   t1[22376] := -0.0600096;
   t1[22377] := -0.0732072;
   t1[22378] := -0.0857643;
   t1[22379] := -0.097705;
   t1[22380] := -0.1090593;
   t1[22381] := -0.1198572;
   t1[22382] := -0.130129;
   t1[22383] := -0.1399046;
   t1[22384] := -0.1492141;
   t1[22385] := -0.1580877;
   t1[22386] := -0.1665554;
   t1[22387] := -0.1746473;
   t1[22388] := -0.1823935;
   t1[22389] := -0.189824;
   t1[22390] := -0.196969;
   t1[22391] := -0.2038585;
   t1[22392] := -0.2105227;
   t1[22393] := -0.2169916;
   t1[22394] := -0.2232952;
   t1[22395] := -0.2294637;
   t1[22396] := -0.2355272;
   t1[22397] := -0.2415041;
   t1[22398] := -0.2473547;
   t1[22399] := -0.2530213;
   w2[0] := 0.3822261;
   w2[1] := 0.6735258;
   w2[2] := 0.4999258;
   w2[3] := 0.0709843;
   w2[4] := 0.4040336;
   w2[5] := -0.3168498;
   w2[6] := -0.5318553;
   w2[7] := -0.3348889;
   w2[8] := 0.5234552;
   w2[9] := 0.3241403;
   w2[10] := -0.6014917;
   w2[11] := -0.2869324;
   w2[12] := -0.0813316;
   w2[13] := 0.2735443;
   w2[14] := -0.5975453;
   w2[15] := -0.3671676;
   w2[16] := 0.1604395;
   w2[17] := 0.6218057;
   w2[18] := -0.535407;
   w2[19] := -0.428839;
   w2[20] := 0.4432988;
   w2[21] := -0.1195226;
   w2[22] := -0.1593684;
   w2[23] := -0.4208567;
   w2[24] := -0.0164311;
   w2[25] := 0.1177106;
   w2[26] := -0.1915699;
   w2[27] := -0.2585908;
   w2[28] := 0.7388805;
   w2[29] := 0.7177937;
   w2[30] := 0.9066412;
   w2[31] := -0.3313666;
   w2[32] := -0.5566195;
   w2[33] := 0.1009696;
   w2[34] := 0.7024983;
   w2[35] := -0.0061407;
   w2[36] := 0.9221094;
   w2[37] := 0.9728315;
   w2[38] := 0.7287791;
   w2[39] := 0.1011917;
   w2[40] := 0.1708561;
   w2[41] := 0.0181266;
   w2[42] := -0.3799455;
   w2[43] := -0.2221509;
   w2[44] := -0.2996568;
   w2[45] := 0.1856399;
   w2[46] := -0.2363337;
   w2[47] := 0.3469633;
   w2[48] := -0.3170906;
   w2[49] := -0.3010724;
   w2[50] := -0.4463713;
   w2[51] := 0.4818622;
   w2[52] := -0.2695292;
   w2[53] := -0.4620254;
   w2[54] := 0.0533027;
   w2[55] := -0.395156;
   w2[56] := 0.0408355;
   w2[57] := -0.2507218;
   w2[58] := 0.0280879;
   w2[59] := 0.0458854;
   w2[60] := -0.0139494;
   w2[61] := 0.0098419;
   w2[62] := -0.4868755;
   w2[63] := 0.1032088;
   w2[64] := 0.1231787;
   w2[65] := 0.5223995;
   w2[66] := 0.4042619;
   w2[67] := 0.2341684;
   w2[68] := -0.2304757;
   w2[69] := 0.0635033;
   w2[70] := -0.3774453;
   w2[71] := -0.4428134;
   w2[72] := -0.0484126;
   w2[73] := 0.2895669;
   w2[74] := -0.6764416;
   w2[75] := -0.3088431;
   w2[76] := 0.4827037;
   w2[77] := 0.0691548;
   w2[78] := 0.4661854;
   w2[79] := 0.1204736;
   w2[80] := -0.4872637;
   w2[81] := -0.0951735;
   w2[82] := -0.0189593;
   w2[83] := -0.1372051;
   w2[84] := -0.9140335;
   w2[85] := -0.8600995;
   w2[86] := -1.056187;
   w2[87] := -0.5128109;
   w2[88] := -0.7898985;
   w2[89] := -0.5083115;
   w2[90] := -0.5282256;
   w2[91] := -0.4263123;
   w2[92] := -1.016044;
   w2[93] := -0.0212463;
   w2[94] := 0.6550046;
   w2[95] := 0.4706961;
   w2[96] := -0.1141442;
   w2[97] := -0.2175039;
   w2[98] := -0.2840221;
   w2[99] := -0.3306261;
   w2[100] := -0.2441688;
   w2[101] := 0.3605514;
   w2[102] := -0.3955784;
   w2[103] := 0.0529358;
   w2[104] := 0.3398173;
   w2[105] := 0.3715278;
   w2[106] := 0.429172;
   w2[107] := 0.4002611;
   w2[108] := -0.2264336;
   w2[109] := 0.312763;
   w2[110] := 0.5647593;
   w2[111] := 0.0224205;
   w2[112] := -0.5216327;
   w2[113] := -0.2093005;
   w2[114] := -0.3824884;
   w2[115] := -0.0496232;
   w2[116] := -0.0204715;
   w2[117] := 0.3446302;
   w2[118] := -0.1566623;
   w2[119] := -0.1314349;
   w2[120] := -0.3364701;
   w2[121] := -0.5365704;
   w2[122] := -0.3706124;
   w2[123] := -0.2384351;
   w2[124] := 0.2599077;
   w2[125] := 0.0878742;
   w2[126] := -0.1167608;
   w2[127] := 0.4445257;
   w2[128] := 0.0472859;
   w2[129] := -0.2039315;
   w2[130] := -0.0123044;
   w2[131] := 0.5347427;
   w2[132] := -0.4565654;
   w2[133] := -0.1309683;
   w2[134] := -0.1916631;
   w2[135] := -0.0229556;
   w2[136] := -0.1463313;
   w2[137] := 0.0884493;
   w2[138] := -0.1268248;
   w2[139] := 0.1727386;
   w2[140] := 0.1864566;
   w2[141] := 0.0450289;
   w2[142] := 0.2544484;
   w2[143] := -0.1416016;
   w2[144] := -0.1781151;
   w2[145] := -0.1914191;
   w2[146] := 0.3022377;
   w2[147] := 0.2656204;
   w2[148] := 0.135544;
   w2[149] := 0.5225624;
   w2[150] := 0.8165789;
   w2[151] := 0.3793563;
   w2[152] := -0.1251971;
   w2[153] := -0.032513;
   w2[154] := -0.1753309;
   w2[155] := -0.429324;
   w2[156] := -0.4619711;
   w2[157] := 0.3961401;
   w2[158] := -0.6358346;
   w2[159] := 0.531637;
   w2[160] := 0.2908633;
   w2[161] := 0.2183272;
   w2[162] := 0.3942987;
   w2[163] := 0.3020125;
   w2[164] := -0.4793546;
   w2[165] := 0.0537859;
   w2[166] := 0.2855184;
   w2[167] := -0.2678719;
   w2[168] := 0.3169011;
   w2[169] := 0.0269058;
   w2[170] := 0.139307;
   w2[171] := 0.2074015;
   w2[172] := 0.044378;
   w2[173] := 0.3336064;
   w2[174] := -0.1919886;
   w2[175] := 0.0043234;
   w2[176] := 0.5604227;
   w2[177] := -0.1127777;
   w2[178] := -0.3165137;
   w2[179] := 0.2200206;
   w2[180] := -0.2163805;
   w2[181] := -0.239696;
   w2[182] := 0.1728129;
   w2[183] := -0.1887252;
   w2[184] := 0.2727011;
   w2[185] := 0.1560453;
   w2[186] := 0.457509;
   w2[187] := -0.2272316;
   w2[188] := 0.3077642;
   w2[189] := 0.06774;
   w2[190] := -0.050842;
   w2[191] := 0.0844207;
   w2[192] := 0.2612096;
   w2[193] := -0.0461612;
   w2[194] := 0.196588;
   w2[195] := 0.1832603;
   w2[196] := -0.1259902;
   w2[197] := 0.4958175;
   w2[198] := 0.3578667;
   w2[199] := -0.2289235;
   w2[200] := 0.0412198;
   w2[201] := -0.1472023;
   w2[202] := 0.5003238;
   w2[203] := 0.2104491;
   w2[204] := -0.3506398;
   w2[205] := -0.7278167;
   w2[206] := -0.1053378;
   w2[207] := -0.6664331;
   w2[208] := 0.3304765;
   w2[209] := 0.1904697;
   w2[210] := -0.5255481;
   w2[211] := 0.3779066;
   w2[212] := 0.575013;
   w2[213] := -0.4405918;
   w2[214] := 0.0437819;
   w2[215] := 0.0799071;
   w2[216] := -0.3873571;
   w2[217] := -0.1107465;
   w2[218] := -0.2144487;
   w2[219] := -0.452094;
   w2[220] := -0.0942226;
   w2[221] := -0.1042965;
   w2[222] := -0.0900685;
   w2[223] := -0.0358909;
   w2[224] := 0.5961101;
   w2[225] := -0.0502036;
   w2[226] := -0.205787;
   w2[227] := 0.1793782;
   w2[228] := 0.0139435;
   w2[229] := 0.140426;
   w2[230] := -0.1710399;
   w2[231] := -0.1097762;
   w2[232] := 0.6955358;
   w2[233] := -0.0941478;
   w2[234] := -0.6882815;
   w2[235] := -0.2339452;
   w2[236] := -0.5887371;
   w2[237] := 0.0302498;
   w2[238] := 0.2707806;
   w2[239] := -0.6653628;
   w2[240] := 0.3887634;
   w2[241] := 0.1627363;
   w2[242] := 0.0122889;
   w2[243] := -0.4034282;
   w2[244] := 0.3380547;
   w2[245] := -0.0177897;
   w2[246] := -0.1635698;
   w2[247] := -0.1298062;
   w2[248] := 0.2896215;
   w2[249] := 0.1131524;
   w2[250] := -0.2054364;
   w2[251] := 0.0131579;
   w2[252] := -0.890228;
   w2[253] := -0.6914336;
   w2[254] := -0.8277874;
   w2[255] := 0.254033;
   w2[256] := 0.179194;
   w2[257] := 0.0266804;
   w2[258] := -0.1867425;
   w2[259] := 0.1680747;
   w2[260] := -1.05107;
   w2[261] := -0.5665534;
   w2[262] := -0.1247267;
   w2[263] := -0.053494;
   w2[264] := 0.23726;
   w2[265] := -0.584154;
   w2[266] := -0.2938985;
   w2[267] := 0.1965791;
   w2[268] := 0.5103638;
   w2[269] := -0.0550255;
   w2[270] := -1.126066;
   w2[271] := 0.0735265;
   w2[272] := -0.2777269;
   w2[273] := 0.3135782;
   w2[274] := 0.1041824;
   w2[275] := -0.1324059;
   w2[276] := -0.3669493;
   w2[277] := -0.2885313;
   w2[278] := -0.367729;
   w2[279] := 0.1541151;
   w2[280] := 0.1346243;
   w2[281] := 0.6931639;
   w2[282] := 0.3574378;
   w2[283] := -0.1421183;
   w2[284] := 0.2825844;
   w2[285] := 0.0992049;
   w2[286] := 0.3324718;
   w2[287] := 0.168798;
   w2[288] := 0.1662632;
   w2[289] := -0.5125447;
   w2[290] := 0.1457812;
   w2[291] := -0.2258452;
   w2[292] := -0.2428768;
   w2[293] := 0.2717957;
   w2[294] := 0.0867224;
   w2[295] := -0.2496022;
   w2[296] := 0.1867056;
   w2[297] := -0.4031086;
   w2[298] := 0.4832774;
   w2[299] := 0.2478154;
   w2[300] := 0.0475016;
   w2[301] := -0.1532699;
   w2[302] := -0.6021184;
   w2[303] := -0.4835578;
   w2[304] := 0.348039;
   w2[305] := -0.0061014;
   w2[306] := 0.2888969;
   w2[307] := 0.0215752;
   w2[308] := 0.0208341;
   w2[309] := 0.5199659;
   w2[310] := 0.3490263;
   w2[311] := -0.0288161;
   w2[312] := -0.068543;
   w2[313] := -0.1182679;
   w2[314] := 0.3420109;
   w2[315] := -0.0353185;
   w2[316] := -0.1071727;
   w2[317] := -0.7671919;
   w2[318] := -0.3097001;
   w2[319] := 0.0119445;
   w2[320] := 0.1677119;
   w2[321] := -0.0187103;
   w2[322] := -0.0632623;
   w2[323] := 0.3558021;
   w2[324] := 0.4361037;
   w2[325] := -0.5477799;
   w2[326] := 0.1640894;
   w2[327] := 0.3476633;
   w2[328] := -0.2296589;
   w2[329] := -0.0005878;
   w2[330] := -0.1486427;
   w2[331] := -0.1145124;
   w2[332] := 0.1935411;
   w2[333] := -0.0498571;
   w2[334] := 0.007102;
   w2[335] := 0.1442345;
   w2[336] := -0.7647343;
   w2[337] := -0.7446802;
   w2[338] := -0.8727151;
   w2[339] := 0.3649753;
   w2[340] := 0.182284;
   w2[341] := 0.2168968;
   w2[342] := -0.3110866;
   w2[343] := 0.2285281;
   w2[344] := -0.8572159;
   w2[345] := -0.253249;
   w2[346] := -0.1099993;
   w2[347] := -0.1176312;
   w2[348] := 0.3110442;
   w2[349] := -0.0493409;
   w2[350] := 0.0371198;
   w2[351] := 0.2336326;
   w2[352] := 0.2238284;
   w2[353] := -0.0283122;
   w2[354] := -0.1704783;
   w2[355] := 0.0574998;
   w2[356] := -0.2733924;
   w2[357] := 0.0665076;
   w2[358] := 0.0320759;
   w2[359] := -0.1596949;
   w2[360] := -0.2385386;
   w2[361] := -0.2472534;
   w2[362] := -0.1323308;
   w2[363] := 0.1628101;
   w2[364] := 0.4503315;
   w2[365] := 0.1501646;
   w2[366] := 0.1143262;
   w2[367] := 0.023902;
   w2[368] := 0.0073025;
   w2[369] := 0.1456288;
   w2[370] := -0.3334046;
   w2[371] := 0.0482971;
   w2[372] := 0.4867398;
   w2[373] := -0.4917139;
   w2[374] := -0.6253324;
   w2[375] := -0.1267435;
   w2[376] := -0.2428251;
   w2[377] := -0.2196695;
   w2[378] := 0.1073758;
   w2[379] := 0.0506342;
   w2[380] := 0.4630886;
   w2[381] := -0.1982542;
   w2[382] := 0.3006389;
   w2[383] := -0.1852189;
   w2[384] := 0.1438557;
   w2[385] := 0.2112408;
   w2[386] := -0.1989525;
   w2[387] := -0.5165743;
   w2[388] := 0.2818699;
   w2[389] := 0.1988503;
   w2[390] := 0.0899179;
   w2[391] := 0.0992274;
   w2[392] := 0.3425773;
   w2[393] := -0.0475926;
   w2[394] := 0.0767343;
   w2[395] := 0.0394692;
   w2[396] := 0.1684201;
   w2[397] := -0.1340467;
   w2[398] := -0.3633062;
   w2[399] := -0.3210598;
   w2[400] := 0.5503753;
   w2[401] := 0.2680424;
   w2[402] := -0.2979992;
   w2[403] := -0.3373846;
   w2[404] := -0.2860682;
   w2[405] := 0.0260232;
   w2[406] := -0.1706583;
   w2[407] := -0.4802254;
   w2[408] := 0.1432097;
   w2[409] := 0.2762946;
   w2[410] := -0.3853753;
   w2[411] := -0.4026088;
   w2[412] := 0.3293981;
   w2[413] := 0.031134;
   w2[414] := 0.1150283;
   w2[415] := 0.032845;
   w2[416] := 0.1377832;
   w2[417] := 0.2112923;
   w2[418] := 0.0084318;
   w2[419] := 0.0693316;
   w2[420] := 0.0293756;
   w2[421] := 0.1045898;
   w2[422] := 0.2854653;
   w2[423] := 0.0997073;
   w2[424] := 0.1003512;
   w2[425] := -0.0351206;
   w2[426] := 0.4399726;
   w2[427] := 0.2780291;
   w2[428] := -0.0804132;
   w2[429] := 0.7397832;
   w2[430] := 0.7269561;
   w2[431] := 0.2094024;
   w2[432] := -0.2141474;
   w2[433] := 0.2012126;
   w2[434] := -0.2318728;
   w2[435] := -0.1762547;
   w2[436] := -0.0704646;
   w2[437] := 0.2301458;
   w2[438] := -0.0323121;
   w2[439] := 0.1872706;
   w2[440] := 0.4350786;
   w2[441] := 0.266441;
   w2[442] := 0.2541361;
   w2[443] := 0.1549129;
   w2[444] := -0.1279981;
   w2[445] := -0.1567508;
   w2[446] := 0.1148285;
   w2[447] := -0.2802774;
   g4[0] := -3.0;
   g4[1] := -2.877551;
   g4[2] := -2.755102;
   g4[3] := -2.632653;
   g4[4] := -2.510204;
   g4[5] := -2.387755;
   g4[6] := -2.265306;
   g4[7] := -2.142857;
   g4[8] := -2.020408;
   g4[9] := -1.897959;
   g4[10] := -1.77551;
   g4[11] := -1.653061;
   g4[12] := -1.530612;
   g4[13] := -1.408163;
   g4[14] := -1.285714;
   g4[15] := -1.163265;
   g4[16] := -1.040816;
   g4[17] := -0.9183673;
   g4[18] := -0.7959184;
   g4[19] := -0.6734694;
   g4[20] := -0.5510204;
   g4[21] := -0.4285714;
   g4[22] := -0.3061224;
   g4[23] := -0.1836735;
   g4[24] := -0.0612245;
   g4[25] := 0.0612245;
   g4[26] := 0.1836735;
   g4[27] := 0.3061224;
   g4[28] := 0.4285714;
   g4[29] := 0.5510204;
   g4[30] := 0.6734694;
   g4[31] := 0.7959184;
   g4[32] := 0.9183673;
   g4[33] := 1.040816;
   g4[34] := 1.163265;
   g4[35] := 1.285714;
   g4[36] := 1.408163;
   g4[37] := 1.530612;
   g4[38] := 1.653061;
   g4[39] := 1.77551;
   g4[40] := 1.897959;
   g4[41] := 2.020408;
   g4[42] := 2.142857;
   g4[43] := 2.265306;
   g4[44] := 2.387755;
   g4[45] := 2.510204;
   g4[46] := 2.632653;
   g4[47] := 2.755102;
   g4[48] := 2.877551;
   g4[49] := 3.0;
   t5[0] := 0.0969458;
   t5[1] := 0.0975005;
   t5[2] := 0.0980442;
   t5[3] := 0.0985769;
   t5[4] := 0.0990984;
   t5[5] := 0.0996084;
   t5[6] := 0.1001068;
   t5[7] := 0.1005933;
   t5[8] := 0.1010678;
   t5[9] := 0.1015302;
   t5[10] := 0.1019801;
   t5[11] := 0.1024174;
   t5[12] := 0.102842;
   t5[13] := 0.1032536;
   t5[14] := 0.1036521;
   t5[15] := 0.1040372;
   t5[16] := 0.1044088;
   t5[17] := 0.1047666;
   t5[18] := 0.1051106;
   t5[19] := 0.1054404;
   t5[20] := 0.105756;
   t5[21] := 0.1060571;
   t5[22] := 0.1063435;
   t5[23] := 0.1066151;
   t5[24] := 0.1068716;
   t5[25] := 0.1071129;
   t5[26] := 0.1073388;
   t5[27] := 0.107549;
   t5[28] := 0.1077435;
   t5[29] := 0.1079219;
   t5[30] := 0.1080842;
   t5[31] := 0.1082301;
   t5[32] := 0.1083595;
   t5[33] := 0.1084721;
   t5[34] := 0.1085678;
   t5[35] := 0.1086466;
   t5[36] := 0.1087088;
   t5[37] := 0.1087546;
   t5[38] := 0.1087841;
   t5[39] := 0.1087976;
   t5[40] := 0.1087953;
   t5[41] := 0.1087774;
   t5[42] := 0.1087441;
   t5[43] := 0.1086956;
   t5[44] := 0.1086322;
   t5[45] := 0.1085539;
   t5[46] := 0.1084611;
   t5[47] := 0.1083539;
   t5[48] := 0.1082325;
   t5[49] := 0.1080972;
   t5[50] := 0.0692292;
   t5[51] := 0.0688175;
   t5[52] := 0.0684027;
   t5[53] := 0.0679847;
   t5[54] := 0.0675634;
   t5[55] := 0.0671384;
   t5[56] := 0.0667096;
   t5[57] := 0.0662769;
   t5[58] := 0.0658399;
   t5[59] := 0.0653986;
   t5[60] := 0.0649527;
   t5[61] := 0.0645021;
   t5[62] := 0.0640465;
   t5[63] := 0.0635857;
   t5[64] := 0.0631196;
   t5[65] := 0.062648;
   t5[66] := 0.0621706;
   t5[67] := 0.0616873;
   t5[68] := 0.0611979;
   t5[69] := 0.0607022;
   t5[70] := 0.0601999;
   t5[71] := 0.059691;
   t5[72] := 0.0591752;
   t5[73] := 0.0586522;
   t5[74] := 0.058122;
   t5[75] := 0.0575843;
   t5[76] := 0.057039;
   t5[77] := 0.0564858;
   t5[78] := 0.0559245;
   t5[79] := 0.055355;
   t5[80] := 0.054777;
   t5[81] := 0.0541904;
   t5[82] := 0.0535949;
   t5[83] := 0.0529904;
   t5[84] := 0.0523768;
   t5[85] := 0.051754;
   t5[86] := 0.0511223;
   t5[87] := 0.050482;
   t5[88] := 0.0498332;
   t5[89] := 0.0491762;
   t5[90] := 0.0485112;
   t5[91] := 0.0478384;
   t5[92] := 0.0471581;
   t5[93] := 0.0464705;
   t5[94] := 0.0457757;
   t5[95] := 0.0450742;
   t5[96] := 0.0443659;
   t5[97] := 0.0436513;
   t5[98] := 0.0429304;
   t5[99] := 0.0422036;
   t5[100] := 0.0769506;
   t5[101] := 0.0760873;
   t5[102] := 0.0752231;
   t5[103] := 0.074358;
   t5[104] := 0.0734922;
   t5[105] := 0.0726259;
   t5[106] := 0.0717593;
   t5[107] := 0.0708925;
   t5[108] := 0.0700258;
   t5[109] := 0.0691593;
   t5[110] := 0.0682932;
   t5[111] := 0.0674276;
   t5[112] := 0.0665628;
   t5[113] := 0.0656989;
   t5[114] := 0.0648361;
   t5[115] := 0.0639746;
   t5[116] := 0.0631145;
   t5[117] := 0.0622561;
   t5[118] := 0.0613995;
   t5[119] := 0.0605449;
   t5[120] := 0.0596924;
   t5[121] := 0.0588422;
   t5[122] := 0.0579946;
   t5[123] := 0.0571497;
   t5[124] := 0.0563077;
   t5[125] := 0.0554687;
   t5[126] := 0.0546329;
   t5[127] := 0.0538006;
   t5[128] := 0.0529718;
   t5[129] := 0.0521468;
   t5[130] := 0.0513257;
   t5[131] := 0.0505087;
   t5[132] := 0.049696;
   t5[133] := 0.0488878;
   t5[134] := 0.0480843;
   t5[135] := 0.0472854;
   t5[136] := 0.0464911;
   t5[137] := 0.0457015;
   t5[138] := 0.0449164;
   t5[139] := 0.0441359;
   t5[140] := 0.0433598;
   t5[141] := 0.0425883;
   t5[142] := 0.0418212;
   t5[143] := 0.0410585;
   t5[144] := 0.0403002;
   t5[145] := 0.0395462;
   t5[146] := 0.0387965;
   t5[147] := 0.0380511;
   t5[148] := 0.03731;
   t5[149] := 0.036573;
   t5[150] := 0.0185666;
   t5[151] := 0.018039;
   t5[152] := 0.0175079;
   t5[153] := 0.0169733;
   t5[154] := 0.0164355;
   t5[155] := 0.0158946;
   t5[156] := 0.0153508;
   t5[157] := 0.0148043;
   t5[158] := 0.0142552;
   t5[159] := 0.0137036;
   t5[160] := 0.0131499;
   t5[161] := 0.012594;
   t5[162] := 0.0120363;
   t5[163] := 0.0114768;
   t5[164] := 0.0109158;
   t5[165] := 0.0103533;
   t5[166] := 0.0097896;
   t5[167] := 0.0092249;
   t5[168] := 0.0086592;
   t5[169] := 0.0080928;
   t5[170] := 0.0075258;
   t5[171] := 0.0069585;
   t5[172] := 0.0063908;
   t5[173] := 0.0058232;
   t5[174] := 0.0052556;
   t5[175] := 0.0046883;
   t5[176] := 0.0041214;
   t5[177] := 0.0035551;
   t5[178] := 0.0029896;
   t5[179] := 0.002425;
   t5[180] := 0.0018615;
   t5[181] := 0.0012993;
   t5[182] := 0.0007385;
   t5[183] := 0.0001793;
   t5[184] := -0.0003781;
   t5[185] := -0.0009336;
   t5[186] := -0.0014869;
   t5[187] := -0.002038;
   t5[188] := -0.0025867;
   t5[189] := -0.0031328;
   t5[190] := -0.0036761;
   t5[191] := -0.0042165;
   t5[192] := -0.0047537;
   t5[193] := -0.0052877;
   t5[194] := -0.0058183;
   t5[195] := -0.0063453;
   t5[196] := -0.0068684;
   t5[197] := -0.0073877;
   t5[198] := -0.0079029;
   t5[199] := -0.0084138;
   t5[200] := -0.0480992;
   t5[201] := -0.0461759;
   t5[202] := -0.0442379;
   t5[203] := -0.0422851;
   t5[204] := -0.0403176;
   t5[205] := -0.0383352;
   t5[206] := -0.0363378;
   t5[207] := -0.0343254;
   t5[208] := -0.0322979;
   t5[209] := -0.0302553;
   t5[210] := -0.0281974;
   t5[211] := -0.0261242;
   t5[212] := -0.0240356;
   t5[213] := -0.0219317;
   t5[214] := -0.0198121;
   t5[215] := -0.017677;
   t5[216] := -0.0155263;
   t5[217] := -0.0133598;
   t5[218] := -0.0111775;
   t5[219] := -0.0089794;
   t5[220] := -0.0067653;
   t5[221] := -0.0045353;
   t5[222] := -0.0022891;
   t5[223] := -2.68E-05;
   t5[224] := 0.0022517;
   t5[225] := 0.0045464;
   t5[226] := 0.0068576;
   t5[227] := 0.0091852;
   t5[228] := 0.0115292;
   t5[229] := 0.0138899;
   t5[230] := 0.0162671;
   t5[231] := 0.0186611;
   t5[232] := 0.0210719;
   t5[233] := 0.0234995;
   t5[234] := 0.025944;
   t5[235] := 0.028405;
   t5[236] := 0.0308823;
   t5[237] := 0.0333751;
   t5[238] := 0.035883;
   t5[239] := 0.0384056;
   t5[240] := 0.0409424;
   t5[241] := 0.0434929;
   t5[242] := 0.0460565;
   t5[243] := 0.0486329;
   t5[244] := 0.0512215;
   t5[245] := 0.0538219;
   t5[246] := 0.0564335;
   t5[247] := 0.059056;
   t5[248] := 0.0616887;
   t5[249] := 0.0643312;
   t5[250] := 0.0416106;
   t5[251] := 0.0407638;
   t5[252] := 0.039913;
   t5[253] := 0.0390582;
   t5[254] := 0.0381993;
   t5[255] := 0.0373361;
   t5[256] := 0.0364686;
   t5[257] := 0.0355967;
   t5[258] := 0.0347203;
   t5[259] := 0.0338393;
   t5[260] := 0.0329536;
   t5[261] := 0.0320632;
   t5[262] := 0.031168;
   t5[263] := 0.0302678;
   t5[264] := 0.0293625;
   t5[265] := 0.0284521;
   t5[266] := 0.0275366;
   t5[267] := 0.0266157;
   t5[268] := 0.0256895;
   t5[269] := 0.0247577;
   t5[270] := 0.0238204;
   t5[271] := 0.0228775;
   t5[272] := 0.0219288;
   t5[273] := 0.0209743;
   t5[274] := 0.0200138;
   t5[275] := 0.0190474;
   t5[276] := 0.0180748;
   t5[277] := 0.0170961;
   t5[278] := 0.0161111;
   t5[279] := 0.0151197;
   t5[280] := 0.0141218;
   t5[281] := 0.0131174;
   t5[282] := 0.0121064;
   t5[283] := 0.0110886;
   t5[284] := 0.0100641;
   t5[285] := 0.0090329;
   t5[286] := 0.0079953;
   t5[287] := 0.0069515;
   t5[288] := 0.005902;
   t5[289] := 0.0048468;
   t5[290] := 0.0037862;
   t5[291] := 0.0027206;
   t5[292] := 0.0016502;
   t5[293] := 0.0005753;
   t5[294] := -0.000504;
   t5[295] := -0.0015873;
   t5[296] := -0.0026743;
   t5[297] := -0.0037649;
   t5[298] := -0.0048587;
   t5[299] := -0.0059555;
   t5[300] := 0.040686;
   t5[301] := 0.0380326;
   t5[302] := 0.0353805;
   t5[303] := 0.0327302;
   t5[304] := 0.0300825;
   t5[305] := 0.0274376;
   t5[306] := 0.0247961;
   t5[307] := 0.0221584;
   t5[308] := 0.0195253;
   t5[309] := 0.016897;
   t5[310] := 0.0142741;
   t5[311] := 0.0116571;
   t5[312] := 0.0090466;
   t5[313] := 0.006443;
   t5[314] := 0.0038467;
   t5[315] := 0.0012584;
   t5[316] := -0.0013215;
   t5[317] := -0.0038925;
   t5[318] := -0.0064541;
   t5[319] := -0.0090057;
   t5[320] := -0.0115469;
   t5[321] := -0.0140773;
   t5[322] := -0.0165961;
   t5[323] := -0.0191031;
   t5[324] := -0.0215977;
   t5[325] := -0.0240793;
   t5[326] := -0.0265474;
   t5[327] := -0.0290017;
   t5[328] := -0.0314415;
   t5[329] := -0.0338664;
   t5[330] := -0.0362759;
   t5[331] := -0.0386694;
   t5[332] := -0.0410465;
   t5[333] := -0.0434067;
   t5[334] := -0.0457494;
   t5[335] := -0.0480745;
   t5[336] := -0.050382;
   t5[337] := -0.0526716;
   t5[338] := -0.0549433;
   t5[339] := -0.0571972;
   t5[340] := -0.059433;
   t5[341] := -0.0616507;
   t5[342] := -0.0638503;
   t5[343] := -0.0660316;
   t5[344] := -0.0681946;
   t5[345] := -0.0703393;
   t5[346] := -0.0724654;
   t5[347] := -0.074573;
   t5[348] := -0.076662;
   t5[349] := -0.0787324;
   t5[350] := 0.0090538;
   t5[351] := 0.00985;
   t5[352] := 0.0106394;
   t5[353] := 0.0114219;
   t5[354] := 0.0121974;
   t5[355] := 0.0129658;
   t5[356] := 0.0137272;
   t5[357] := 0.0144813;
   t5[358] := 0.0152283;
   t5[359] := 0.015968;
   t5[360] := 0.0167005;
   t5[361] := 0.0174255;
   t5[362] := 0.0181432;
   t5[363] := 0.0188533;
   t5[364] := 0.019556;
   t5[365] := 0.020251;
   t5[366] := 0.0209385;
   t5[367] := 0.0216182;
   t5[368] := 0.0222903;
   t5[369] := 0.0229545;
   t5[370] := 0.0236109;
   t5[371] := 0.0242594;
   t5[372] := 0.0248999;
   t5[373] := 0.0255325;
   t5[374] := 0.026157;
   t5[375] := 0.0267733;
   t5[376] := 0.0273816;
   t5[377] := 0.0279816;
   t5[378] := 0.0285733;
   t5[379] := 0.0291567;
   t5[380] := 0.0297317;
   t5[381] := 0.0302983;
   t5[382] := 0.0308565;
   t5[383] := 0.0314061;
   t5[384] := 0.0319471;
   t5[385] := 0.0324795;
   t5[386] := 0.0330033;
   t5[387] := 0.0335185;
   t5[388] := 0.0340251;
   t5[389] := 0.0345232;
   t5[390] := 0.0350126;
   t5[391] := 0.0354935;
   t5[392] := 0.0359658;
   t5[393] := 0.0364295;
   t5[394] := 0.0368846;
   t5[395] := 0.0373312;
   t5[396] := 0.0377692;
   t5[397] := 0.0381986;
   t5[398] := 0.0386195;
   t5[399] := 0.0390318;
   t5[400] := 0.0821998;
   t5[401] := 0.0816142;
   t5[402] := 0.0810245;
   t5[403] := 0.0804307;
   t5[404] := 0.0798329;
   t5[405] := 0.0792312;
   t5[406] := 0.0786256;
   t5[407] := 0.0780161;
   t5[408] := 0.0774028;
   t5[409] := 0.0767859;
   t5[410] := 0.0761652;
   t5[411] := 0.075541;
   t5[412] := 0.0749132;
   t5[413] := 0.074282;
   t5[414] := 0.0736473;
   t5[415] := 0.0730093;
   t5[416] := 0.0723679;
   t5[417] := 0.0717234;
   t5[418] := 0.0710756;
   t5[419] := 0.0704247;
   t5[420] := 0.0697708;
   t5[421] := 0.0691138;
   t5[422] := 0.0684539;
   t5[423] := 0.0677911;
   t5[424] := 0.0671255;
   t5[425] := 0.0664571;
   t5[426] := 0.065786;
   t5[427] := 0.0651122;
   t5[428] := 0.0644359;
   t5[429] := 0.063757;
   t5[430] := 0.0630756;
   t5[431] := 0.0623918;
   t5[432] := 0.0617057;
   t5[433] := 0.0610173;
   t5[434] := 0.0603267;
   t5[435] := 0.0596339;
   t5[436] := 0.0589391;
   t5[437] := 0.0582424;
   t5[438] := 0.057544;
   t5[439] := 0.0568439;
   t5[440] := 0.0561423;
   t5[441] := 0.0554394;
   t5[442] := 0.0547352;
   t5[443] := 0.0540298;
   t5[444] := 0.0533235;
   t5[445] := 0.0526162;
   t5[446] := 0.0519082;
   t5[447] := 0.0511996;
   t5[448] := 0.0504905;
   t5[449] := 0.049781;
   t5[450] := -0.0523619;
   t5[451] := -0.0515334;
   t5[452] := -0.050693;
   t5[453] := -0.0498403;
   t5[454] := -0.0489752;
   t5[455] := -0.0480973;
   t5[456] := -0.0472064;
   t5[457] := -0.0463022;
   t5[458] := -0.0453845;
   t5[459] := -0.044453;
   t5[460] := -0.0435074;
   t5[461] := -0.0425475;
   t5[462] := -0.041573;
   t5[463] := -0.0405836;
   t5[464] := -0.0395791;
   t5[465] := -0.0385592;
   t5[466] := -0.0375237;
   t5[467] := -0.0364722;
   t5[468] := -0.0354045;
   t5[469] := -0.0343204;
   t5[470] := -0.0332196;
   t5[471] := -0.0321018;
   t5[472] := -0.0309667;
   t5[473] := -0.0298141;
   t5[474] := -0.0286438;
   t5[475] := -0.0274554;
   t5[476] := -0.0262487;
   t5[477] := -0.0250234;
   t5[478] := -0.0237793;
   t5[479] := -0.0225161;
   t5[480] := -0.0212336;
   t5[481] := -0.0199314;
   t5[482] := -0.0186093;
   t5[483] := -0.017267;
   t5[484] := -0.0159044;
   t5[485] := -0.0145215;
   t5[486] := -0.0131187;
   t5[487] := -0.0116963;
   t5[488] := -0.0102548;
   t5[489] := -0.0087943;
   t5[490] := -0.0073153;
   t5[491] := -0.0058181;
   t5[492] := -0.004303;
   t5[493] := -0.0027705;
   t5[494] := -0.0012208;
   t5[495] := 0.0003458;
   t5[496] := 0.0019288;
   t5[497] := 0.0035279;
   t5[498] := 0.0051428;
   t5[499] := 0.0067732;
   t5[500] := 0.0102707;
   t5[501] := 0.0091437;
   t5[502] := 0.0080237;
   t5[503] := 0.0069108;
   t5[504] := 0.0058052;
   t5[505] := 0.0047069;
   t5[506] := 0.0036161;
   t5[507] := 0.0025329;
   t5[508] := 0.0014575;
   t5[509] := 0.00039;
   t5[510] := -0.0006694;
   t5[511] := -0.0017207;
   t5[512] := -0.0027637;
   t5[513] := -0.0037982;
   t5[514] := -0.0048241;
   t5[515] := -0.0058414;
   t5[516] := -0.0068497;
   t5[517] := -0.0078491;
   t5[518] := -0.0088394;
   t5[519] := -0.0098204;
   t5[520] := -0.010792;
   t5[521] := -0.0117542;
   t5[522] := -0.0127066;
   t5[523] := -0.0136493;
   t5[524] := -0.014582;
   t5[525] := -0.0155047;
   t5[526] := -0.0164172;
   t5[527] := -0.0173193;
   t5[528] := -0.018211;
   t5[529] := -0.0190921;
   t5[530] := -0.0199625;
   t5[531] := -0.020822;
   t5[532] := -0.0216705;
   t5[533] := -0.0225078;
   t5[534] := -0.0233339;
   t5[535] := -0.0241488;
   t5[536] := -0.0249524;
   t5[537] := -0.0257448;
   t5[538] := -0.0265261;
   t5[539] := -0.0272963;
   t5[540] := -0.0280555;
   t5[541] := -0.0288037;
   t5[542] := -0.029541;
   t5[543] := -0.0302674;
   t5[544] := -0.0309829;
   t5[545] := -0.0316877;
   t5[546] := -0.0323817;
   t5[547] := -0.0330651;
   t5[548] := -0.0337378;
   t5[549] := -0.0344;
   t5[550] := 0.0980121;
   t5[551] := 0.0984799;
   t5[552] := 0.0989301;
   t5[553] := 0.0993623;
   t5[554] := 0.0997762;
   t5[555] := 0.1001716;
   t5[556] := 0.1005483;
   t5[557] := 0.1009058;
   t5[558] := 0.101244;
   t5[559] := 0.1015626;
   t5[560] := 0.1018612;
   t5[561] := 0.1021396;
   t5[562] := 0.1023975;
   t5[563] := 0.1026347;
   t5[564] := 0.1028509;
   t5[565] := 0.1030457;
   t5[566] := 0.103219;
   t5[567] := 0.1033703;
   t5[568] := 0.1034995;
   t5[569] := 0.1036062;
   t5[570] := 0.1036903;
   t5[571] := 0.1037513;
   t5[572] := 0.1037891;
   t5[573] := 0.1038033;
   t5[574] := 0.1037937;
   t5[575] := 0.1037599;
   t5[576] := 0.1037018;
   t5[577] := 0.103619;
   t5[578] := 0.1035112;
   t5[579] := 0.1033782;
   t5[580] := 0.1032197;
   t5[581] := 0.1030353;
   t5[582] := 0.102825;
   t5[583] := 0.1025882;
   t5[584] := 0.1023249;
   t5[585] := 0.102035;
   t5[586] := 0.101719;
   t5[587] := 0.101377;
   t5[588] := 0.1010094;
   t5[589] := 0.1006164;
   t5[590] := 0.1001984;
   t5[591] := 0.0997556;
   t5[592] := 0.0992884;
   t5[593] := 0.0987969;
   t5[594] := 0.0982816;
   t5[595] := 0.0977427;
   t5[596] := 0.0971805;
   t5[597] := 0.0965953;
   t5[598] := 0.0959873;
   t5[599] := 0.095357;
   t5[600] := -0.0973992;
   t5[601] := -0.0965358;
   t5[602] := -0.0956592;
   t5[603] := -0.0947693;
   t5[604] := -0.0938661;
   t5[605] := -0.0929496;
   t5[606] := -0.0920197;
   t5[607] := -0.0910766;
   t5[608] := -0.0901201;
   t5[609] := -0.0891502;
   t5[610] := -0.088167;
   t5[611] := -0.0871704;
   t5[612] := -0.0861604;
   t5[613] := -0.0851371;
   t5[614] := -0.0841003;
   t5[615] := -0.0830502;
   t5[616] := -0.0819866;
   t5[617] := -0.0809096;
   t5[618] := -0.0798191;
   t5[619] := -0.0787152;
   t5[620] := -0.0775978;
   t5[621] := -0.076467;
   t5[622] := -0.0753226;
   t5[623] := -0.0741648;
   t5[624] := -0.0729935;
   t5[625] := -0.0718087;
   t5[626] := -0.0706103;
   t5[627] := -0.0693984;
   t5[628] := -0.068173;
   t5[629] := -0.066934;
   t5[630] := -0.0656814;
   t5[631] := -0.0644153;
   t5[632] := -0.0631355;
   t5[633] := -0.0618422;
   t5[634] := -0.0605353;
   t5[635] := -0.059215;
   t5[636] := -0.0578814;
   t5[637] := -0.0565348;
   t5[638] := -0.0551754;
   t5[639] := -0.0538035;
   t5[640] := -0.0524192;
   t5[641] := -0.0510228;
   t5[642] := -0.0496145;
   t5[643] := -0.0481946;
   t5[644] := -0.0467632;
   t5[645] := -0.0453206;
   t5[646] := -0.043867;
   t5[647] := -0.0424026;
   t5[648] := -0.0409276;
   t5[649] := -0.0394423;
   t5[650] := 0.0479108;
   t5[651] := 0.0474616;
   t5[652] := 0.0470249;
   t5[653] := 0.046601;
   t5[654] := 0.0461899;
   t5[655] := 0.0457921;
   t5[656] := 0.0454076;
   t5[657] := 0.0450368;
   t5[658] := 0.0446799;
   t5[659] := 0.0443371;
   t5[660] := 0.0440086;
   t5[661] := 0.0436947;
   t5[662] := 0.0433956;
   t5[663] := 0.0431116;
   t5[664] := 0.0428428;
   t5[665] := 0.0425895;
   t5[666] := 0.0423519;
   t5[667] := 0.0421303;
   t5[668] := 0.041925;
   t5[669] := 0.041736;
   t5[670] := 0.0415637;
   t5[671] := 0.0414083;
   t5[672] := 0.04127;
   t5[673] := 0.0411491;
   t5[674] := 0.0410458;
   t5[675] := 0.0409603;
   t5[676] := 0.0408929;
   t5[677] := 0.0408437;
   t5[678] := 0.0408131;
   t5[679] := 0.0408012;
   t5[680] := 0.0408083;
   t5[681] := 0.0408346;
   t5[682] := 0.0408804;
   t5[683] := 0.0409459;
   t5[684] := 0.0410312;
   t5[685] := 0.0411363;
   t5[686] := 0.0412607;
   t5[687] := 0.041404;
   t5[688] := 0.0415658;
   t5[689] := 0.0417459;
   t5[690] := 0.0419438;
   t5[691] := 0.042159;
   t5[692] := 0.0423913;
   t5[693] := 0.0426403;
   t5[694] := 0.0429055;
   t5[695] := 0.0431867;
   t5[696] := 0.0434833;
   t5[697] := 0.043795;
   t5[698] := 0.0441216;
   t5[699] := 0.0444624;
   t5[700] := 0.1111941;
   t5[701] := 0.110256;
   t5[702] := 0.1093125;
   t5[703] := 0.1083636;
   t5[704] := 0.1074093;
   t5[705] := 0.1064497;
   t5[706] := 0.1054847;
   t5[707] := 0.1045146;
   t5[708] := 0.1035392;
   t5[709] := 0.1025586;
   t5[710] := 0.1015728;
   t5[711] := 0.100582;
   t5[712] := 0.0995861;
   t5[713] := 0.0985852;
   t5[714] := 0.0975793;
   t5[715] := 0.0965685;
   t5[716] := 0.0955527;
   t5[717] := 0.0945321;
   t5[718] := 0.0935066;
   t5[719] := 0.0924763;
   t5[720] := 0.0914413;
   t5[721] := 0.0904016;
   t5[722] := 0.0893572;
   t5[723] := 0.0883082;
   t5[724] := 0.0872545;
   t5[725] := 0.0861963;
   t5[726] := 0.0851335;
   t5[727] := 0.0840663;
   t5[728] := 0.0829947;
   t5[729] := 0.0819186;
   t5[730] := 0.0808382;
   t5[731] := 0.0797534;
   t5[732] := 0.0786643;
   t5[733] := 0.077571;
   t5[734] := 0.0764735;
   t5[735] := 0.0753718;
   t5[736] := 0.074266;
   t5[737] := 0.0731561;
   t5[738] := 0.0720422;
   t5[739] := 0.0709243;
   t5[740] := 0.0698024;
   t5[741] := 0.0686767;
   t5[742] := 0.0675472;
   t5[743] := 0.0664139;
   t5[744] := 0.0652768;
   t5[745] := 0.0641361;
   t5[746] := 0.0629917;
   t5[747] := 0.0618438;
   t5[748] := 0.0606922;
   t5[749] := 0.0595373;
   t5[750] := -0.0148444;
   t5[751] := -0.0159877;
   t5[752] := -0.0171278;
   t5[753] := -0.0182647;
   t5[754] := -0.0193983;
   t5[755] := -0.0205285;
   t5[756] := -0.0216554;
   t5[757] := -0.0227787;
   t5[758] := -0.0238985;
   t5[759] := -0.0250145;
   t5[760] := -0.0261269;
   t5[761] := -0.0272354;
   t5[762] := -0.0283401;
   t5[763] := -0.0294408;
   t5[764] := -0.0305375;
   t5[765] := -0.03163;
   t5[766] := -0.0327184;
   t5[767] := -0.0338025;
   t5[768] := -0.0348823;
   t5[769] := -0.0359576;
   t5[770] := -0.0370284;
   t5[771] := -0.0380947;
   t5[772] := -0.0391564;
   t5[773] := -0.0402133;
   t5[774] := -0.0412654;
   t5[775] := -0.0423127;
   t5[776] := -0.043355;
   t5[777] := -0.0443923;
   t5[778] := -0.0454244;
   t5[779] := -0.0464514;
   t5[780] := -0.0474732;
   t5[781] := -0.0484896;
   t5[782] := -0.0495007;
   t5[783] := -0.0505062;
   t5[784] := -0.0515062;
   t5[785] := -0.0525006;
   t5[786] := -0.0534895;
   t5[787] := -0.0544727;
   t5[788] := -0.0554504;
   t5[789] := -0.0564225;
   t5[790] := -0.0573889;
   t5[791] := -0.0583498;
   t5[792] := -0.0593051;
   t5[793] := -0.0602548;
   t5[794] := -0.0611989;
   t5[795] := -0.0621374;
   t5[796] := -0.0630702;
   t5[797] := -0.0639975;
   t5[798] := -0.0649191;
   t5[799] := -0.0658352;
   t5[800] := 0.1048705;
   t5[801] := 0.1049797;
   t5[802] := 0.105091;
   t5[803] := 0.1052044;
   t5[804] := 0.1053198;
   t5[805] := 0.1054372;
   t5[806] := 0.1055567;
   t5[807] := 0.1056781;
   t5[808] := 0.1058014;
   t5[809] := 0.1059267;
   t5[810] := 0.1060538;
   t5[811] := 0.1061828;
   t5[812] := 0.1063137;
   t5[813] := 0.1064463;
   t5[814] := 0.1065808;
   t5[815] := 0.106717;
   t5[816] := 0.1068549;
   t5[817] := 0.1069946;
   t5[818] := 0.107136;
   t5[819] := 0.107279;
   t5[820] := 0.1074236;
   t5[821] := 0.1075699;
   t5[822] := 0.1077177;
   t5[823] := 0.1078672;
   t5[824] := 0.1080181;
   t5[825] := 0.1081705;
   t5[826] := 0.1083245;
   t5[827] := 0.1084799;
   t5[828] := 0.1086367;
   t5[829] := 0.1087949;
   t5[830] := 0.1089545;
   t5[831] := 0.1091155;
   t5[832] := 0.1092778;
   t5[833] := 0.1094414;
   t5[834] := 0.1096063;
   t5[835] := 0.1097724;
   t5[836] := 0.1099396;
   t5[837] := 0.1101077;
   t5[838] := 0.1102767;
   t5[839] := 0.1104465;
   t5[840] := 0.1106169;
   t5[841] := 0.1107879;
   t5[842] := 0.1109593;
   t5[843] := 0.111131;
   t5[844] := 0.1113029;
   t5[845] := 0.111475;
   t5[846] := 0.111647;
   t5[847] := 0.1118189;
   t5[848] := 0.1119906;
   t5[849] := 0.112162;
   t5[850] := 0.110168;
   t5[851] := 0.1094275;
   t5[852] := 0.1086676;
   t5[853] := 0.1078883;
   t5[854] := 0.1070894;
   t5[855] := 0.1062709;
   t5[856] := 0.1054325;
   t5[857] := 0.1045742;
   t5[858] := 0.1036959;
   t5[859] := 0.1027974;
   t5[860] := 0.1018787;
   t5[861] := 0.1009397;
   t5[862] := 0.0999802;
   t5[863] := 0.0990002;
   t5[864] := 0.0979995;
   t5[865] := 0.096978;
   t5[866] := 0.0959356;
   t5[867] := 0.0948722;
   t5[868] := 0.0937877;
   t5[869] := 0.0926819;
   t5[870] := 0.0915549;
   t5[871] := 0.0904064;
   t5[872] := 0.0892363;
   t5[873] := 0.0880446;
   t5[874] := 0.0868311;
   t5[875] := 0.0855958;
   t5[876] := 0.0843385;
   t5[877] := 0.083059;
   t5[878] := 0.0817574;
   t5[879] := 0.0804334;
   t5[880] := 0.0790871;
   t5[881] := 0.0777182;
   t5[882] := 0.0763266;
   t5[883] := 0.0749123;
   t5[884] := 0.0734752;
   t5[885] := 0.0720154;
   t5[886] := 0.0705333;
   t5[887] := 0.0690293;
   t5[888] := 0.0675037;
   t5[889] := 0.0659568;
   t5[890] := 0.0643889;
   t5[891] := 0.0628005;
   t5[892] := 0.0611919;
   t5[893] := 0.0595634;
   t5[894] := 0.0579154;
   t5[895] := 0.0562482;
   t5[896] := 0.0545621;
   t5[897] := 0.0528576;
   t5[898] := 0.0511348;
   t5[899] := 0.0493943;
   t5[900] := 0.0740068;
   t5[901] := 0.0736119;
   t5[902] := 0.0732176;
   t5[903] := 0.0728238;
   t5[904] := 0.0724307;
   t5[905] := 0.0720383;
   t5[906] := 0.0716467;
   t5[907] := 0.0712559;
   t5[908] := 0.070866;
   t5[909] := 0.0704771;
   t5[910] := 0.0700892;
   t5[911] := 0.0697024;
   t5[912] := 0.0693167;
   t5[913] := 0.0689323;
   t5[914] := 0.0685491;
   t5[915] := 0.0681673;
   t5[916] := 0.0677868;
   t5[917] := 0.0674078;
   t5[918] := 0.0670304;
   t5[919] := 0.0666545;
   t5[920] := 0.0662803;
   t5[921] := 0.0659077;
   t5[922] := 0.065537;
   t5[923] := 0.0651681;
   t5[924] := 0.064801;
   t5[925] := 0.064436;
   t5[926] := 0.0640729;
   t5[927] := 0.0637119;
   t5[928] := 0.0633531;
   t5[929] := 0.0629965;
   t5[930] := 0.0626421;
   t5[931] := 0.0622901;
   t5[932] := 0.0619404;
   t5[933] := 0.0615932;
   t5[934] := 0.0612486;
   t5[935] := 0.0609064;
   t5[936] := 0.0605666;
   t5[937] := 0.0602291;
   t5[938] := 0.059894;
   t5[939] := 0.0595611;
   t5[940] := 0.0592303;
   t5[941] := 0.0589017;
   t5[942] := 0.058575;
   t5[943] := 0.0582504;
   t5[944] := 0.0579276;
   t5[945] := 0.0576066;
   t5[946] := 0.0572875;
   t5[947] := 0.05697;
   t5[948] := 0.0566541;
   t5[949] := 0.0563398;
   t5[950] := 0.0339974;
   t5[951] := 0.0325148;
   t5[952] := 0.0310309;
   t5[953] := 0.0295458;
   t5[954] := 0.0280596;
   t5[955] := 0.0265724;
   t5[956] := 0.0250841;
   t5[957] := 0.023595;
   t5[958] := 0.022105;
   t5[959] := 0.0206144;
   t5[960] := 0.019123;
   t5[961] := 0.0176311;
   t5[962] := 0.0161387;
   t5[963] := 0.0146458;
   t5[964] := 0.0131526;
   t5[965] := 0.0116591;
   t5[966] := 0.0101655;
   t5[967] := 0.0086717;
   t5[968] := 0.0071779;
   t5[969] := 0.0056841;
   t5[970] := 0.0041905;
   t5[971] := 0.0026971;
   t5[972] := 0.001204;
   t5[973] := -0.0002888;
   t5[974] := -0.0017812;
   t5[975] := -0.003273;
   t5[976] := -0.0047642;
   t5[977] := -0.0062548;
   t5[978] := -0.0077446;
   t5[979] := -0.0092335;
   t5[980] := -0.0107216;
   t5[981] := -0.0122086;
   t5[982] := -0.0136946;
   t5[983] := -0.0151795;
   t5[984] := -0.0166631;
   t5[985] := -0.0181454;
   t5[986] := -0.0196262;
   t5[987] := -0.0211054;
   t5[988] := -0.0225829;
   t5[989] := -0.0240585;
   t5[990] := -0.0255321;
   t5[991] := -0.0270036;
   t5[992] := -0.0284728;
   t5[993] := -0.0299397;
   t5[994] := -0.031404;
   t5[995] := -0.0328657;
   t5[996] := -0.0343246;
   t5[997] := -0.0357806;
   t5[998] := -0.0372336;
   t5[999] := -0.0386833;
   t5[1000] := 0.0620911;
   t5[1001] := 0.06173;
   t5[1002] := 0.0613443;
   t5[1003] := 0.0609338;
   t5[1004] := 0.0604981;
   t5[1005] := 0.0600372;
   t5[1006] := 0.0595508;
   t5[1007] := 0.0590387;
   t5[1008] := 0.0585008;
   t5[1009] := 0.0579369;
   t5[1010] := 0.0573467;
   t5[1011] := 0.0567301;
   t5[1012] := 0.0560869;
   t5[1013] := 0.0554168;
   t5[1014] := 0.0547198;
   t5[1015] := 0.0539956;
   t5[1016] := 0.053244;
   t5[1017] := 0.0524647;
   t5[1018] := 0.0516578;
   t5[1019] := 0.0508228;
   t5[1020] := 0.0499597;
   t5[1021] := 0.0490683;
   t5[1022] := 0.0481483;
   t5[1023] := 0.0471996;
   t5[1024] := 0.0462219;
   t5[1025] := 0.0452151;
   t5[1026] := 0.044179;
   t5[1027] := 0.0431134;
   t5[1028] := 0.0420181;
   t5[1029] := 0.0408929;
   t5[1030] := 0.0397376;
   t5[1031] := 0.0385521;
   t5[1032] := 0.0373361;
   t5[1033] := 0.0360894;
   t5[1034] := 0.0348119;
   t5[1035] := 0.0335039;
   t5[1036] := 0.0321659;
   t5[1037] := 0.0307985;
   t5[1038] := 0.0294022;
   t5[1039] := 0.0279776;
   t5[1040] := 0.0265253;
   t5[1041] := 0.0250457;
   t5[1042] := 0.0235394;
   t5[1043] := 0.0220071;
   t5[1044] := 0.0204491;
   t5[1045] := 0.0188661;
   t5[1046] := 0.0172586;
   t5[1047] := 0.0156273;
   t5[1048] := 0.0139725;
   t5[1049] := 0.0122949;
   t5[1050] := 0.1065427;
   t5[1051] := 0.1067164;
   t5[1052] := 0.1068801;
   t5[1053] := 0.1070337;
   t5[1054] := 0.1071769;
   t5[1055] := 0.1073097;
   t5[1056] := 0.1074318;
   t5[1057] := 0.1075431;
   t5[1058] := 0.1076434;
   t5[1059] := 0.1077325;
   t5[1060] := 0.1078104;
   t5[1061] := 0.1078768;
   t5[1062] := 0.1079315;
   t5[1063] := 0.1079745;
   t5[1064] := 0.1080055;
   t5[1065] := 0.1080245;
   t5[1066] := 0.1080311;
   t5[1067] := 0.1080253;
   t5[1068] := 0.1080069;
   t5[1069] := 0.1079757;
   t5[1070] := 0.1079317;
   t5[1071] := 0.1078745;
   t5[1072] := 0.1078041;
   t5[1073] := 0.1077203;
   t5[1074] := 0.1076229;
   t5[1075] := 0.1075117;
   t5[1076] := 0.1073867;
   t5[1077] := 0.1072476;
   t5[1078] := 0.1070943;
   t5[1079] := 0.1069266;
   t5[1080] := 0.1067444;
   t5[1081] := 0.1065475;
   t5[1082] := 0.1063357;
   t5[1083] := 0.1061088;
   t5[1084] := 0.1058668;
   t5[1085] := 0.1056096;
   t5[1086] := 0.1053374;
   t5[1087] := 0.1050503;
   t5[1088] := 0.1047483;
   t5[1089] := 0.1044316;
   t5[1090] := 0.1041004;
   t5[1091] := 0.1037546;
   t5[1092] := 0.1033945;
   t5[1093] := 0.1030202;
   t5[1094] := 0.1026317;
   t5[1095] := 0.1022292;
   t5[1096] := 0.1018128;
   t5[1097] := 0.1013825;
   t5[1098] := 0.1009386;
   t5[1099] := 0.1004812;
   t5[1100] := -0.0022573;
   t5[1101] := -0.0013202;
   t5[1102] := -0.0003888;
   t5[1103] := 0.0005364;
   t5[1104] := 0.0014554;
   t5[1105] := 0.0023679;
   t5[1106] := 0.0032735;
   t5[1107] := 0.0041721;
   t5[1108] := 0.0050634;
   t5[1109] := 0.0059471;
   t5[1110] := 0.006823;
   t5[1111] := 0.0076908;
   t5[1112] := 0.0085503;
   t5[1113] := 0.0094012;
   t5[1114] := 0.0102434;
   t5[1115] := 0.0110764;
   t5[1116] := 0.0119001;
   t5[1117] := 0.0127141;
   t5[1118] := 0.0135184;
   t5[1119] := 0.0143125;
   t5[1120] := 0.0150963;
   t5[1121] := 0.0158695;
   t5[1122] := 0.0166319;
   t5[1123] := 0.0173831;
   t5[1124] := 0.0181229;
   t5[1125] := 0.0188512;
   t5[1126] := 0.0195675;
   t5[1127] := 0.0202718;
   t5[1128] := 0.0209636;
   t5[1129] := 0.0216428;
   t5[1130] := 0.0223092;
   t5[1131] := 0.0229623;
   t5[1132] := 0.0236021;
   t5[1133] := 0.0242283;
   t5[1134] := 0.0248406;
   t5[1135] := 0.025439;
   t5[1136] := 0.0260238;
   t5[1137] := 0.0265951;
   t5[1138] := 0.0271532;
   t5[1139] := 0.0276982;
   t5[1140] := 0.0282303;
   t5[1141] := 0.0287497;
   t5[1142] := 0.0292566;
   t5[1143] := 0.0297512;
   t5[1144] := 0.0302336;
   t5[1145] := 0.0307042;
   t5[1146] := 0.031163;
   t5[1147] := 0.0316102;
   t5[1148] := 0.0320461;
   t5[1149] := 0.0324708;
   t5[1150] := 0.0238222;
   t5[1151] := 0.0241228;
   t5[1152] := 0.0244266;
   t5[1153] := 0.0247341;
   t5[1154] := 0.0250453;
   t5[1155] := 0.0253606;
   t5[1156] := 0.0256802;
   t5[1157] := 0.0260044;
   t5[1158] := 0.0263334;
   t5[1159] := 0.0266675;
   t5[1160] := 0.0270069;
   t5[1161] := 0.0273518;
   t5[1162] := 0.0277027;
   t5[1163] := 0.0280596;
   t5[1164] := 0.0284228;
   t5[1165] := 0.0287926;
   t5[1166] := 0.0291693;
   t5[1167] := 0.029553;
   t5[1168] := 0.0299441;
   t5[1169] := 0.0303428;
   t5[1170] := 0.0307494;
   t5[1171] := 0.031164;
   t5[1172] := 0.031587;
   t5[1173] := 0.0320187;
   t5[1174] := 0.0324591;
   t5[1175] := 0.0329087;
   t5[1176] := 0.0333677;
   t5[1177] := 0.0338362;
   t5[1178] := 0.0343147;
   t5[1179] := 0.0348032;
   t5[1180] := 0.0353021;
   t5[1181] := 0.0358117;
   t5[1182] := 0.0363321;
   t5[1183] := 0.0368637;
   t5[1184] := 0.0374066;
   t5[1185] := 0.0379608;
   t5[1186] := 0.038526;
   t5[1187] := 0.0391019;
   t5[1188] := 0.0396884;
   t5[1189] := 0.040285;
   t5[1190] := 0.0408917;
   t5[1191] := 0.0415081;
   t5[1192] := 0.0421339;
   t5[1193] := 0.042769;
   t5[1194] := 0.0434129;
   t5[1195] := 0.0440656;
   t5[1196] := 0.0447267;
   t5[1197] := 0.045396;
   t5[1198] := 0.0460732;
   t5[1199] := 0.046758;
   t5[1200] := 0.0368159;
   t5[1201] := 0.0383159;
   t5[1202] := 0.0398196;
   t5[1203] := 0.0413271;
   t5[1204] := 0.0428381;
   t5[1205] := 0.0443528;
   t5[1206] := 0.045871;
   t5[1207] := 0.0473928;
   t5[1208] := 0.048918;
   t5[1209] := 0.0504465;
   t5[1210] := 0.0519785;
   t5[1211] := 0.0535137;
   t5[1212] := 0.0550522;
   t5[1213] := 0.0565939;
   t5[1214] := 0.0581387;
   t5[1215] := 0.0596867;
   t5[1216] := 0.0612377;
   t5[1217] := 0.0627918;
   t5[1218] := 0.0643488;
   t5[1219] := 0.0659087;
   t5[1220] := 0.0674714;
   t5[1221] := 0.069037;
   t5[1222] := 0.0706054;
   t5[1223] := 0.0721764;
   t5[1224] := 0.0737502;
   t5[1225] := 0.0753265;
   t5[1226] := 0.0769054;
   t5[1227] := 0.0784869;
   t5[1228] := 0.0800708;
   t5[1229] := 0.0816571;
   t5[1230] := 0.0832458;
   t5[1231] := 0.0848369;
   t5[1232] := 0.0864302;
   t5[1233] := 0.0880257;
   t5[1234] := 0.0896234;
   t5[1235] := 0.0912231;
   t5[1236] := 0.0928247;
   t5[1237] := 0.0944278;
   t5[1238] := 0.0960323;
   t5[1239] := 0.097638;
   t5[1240] := 0.0992446;
   t5[1241] := 0.1008521;
   t5[1242] := 0.1024601;
   t5[1243] := 0.1040684;
   t5[1244] := 0.1056769;
   t5[1245] := 0.1072853;
   t5[1246] := 0.1088935;
   t5[1247] := 0.1105011;
   t5[1248] := 0.1121081;
   t5[1249] := 0.1137142;
   t5[1250] := 0.006496;
   t5[1251] := 0.0056572;
   t5[1252] := 0.0048168;
   t5[1253] := 0.0039752;
   t5[1254] := 0.0031325;
   t5[1255] := 0.0022891;
   t5[1256] := 0.0014451;
   t5[1257] := 0.0006008;
   t5[1258] := -0.0002436;
   t5[1259] := -0.0010878;
   t5[1260] := -0.0019317;
   t5[1261] := -0.002775;
   t5[1262] := -0.0036174;
   t5[1263] := -0.0044587;
   t5[1264] := -0.0052987;
   t5[1265] := -0.0061372;
   t5[1266] := -0.0069739;
   t5[1267] := -0.0078086;
   t5[1268] := -0.008641;
   t5[1269] := -0.0094709;
   t5[1270] := -0.0102982;
   t5[1271] := -0.0111224;
   t5[1272] := -0.0119435;
   t5[1273] := -0.0127612;
   t5[1274] := -0.0135753;
   t5[1275] := -0.0143854;
   t5[1276] := -0.0151914;
   t5[1277] := -0.0159931;
   t5[1278] := -0.0167902;
   t5[1279] := -0.0175825;
   t5[1280] := -0.0183697;
   t5[1281] := -0.0191516;
   t5[1282] := -0.019928;
   t5[1283] := -0.0206987;
   t5[1284] := -0.0214634;
   t5[1285] := -0.0222221;
   t5[1286] := -0.0229749;
   t5[1287] := -0.0237218;
   t5[1288] := -0.0244629;
   t5[1289] := -0.0251984;
   t5[1290] := -0.0259282;
   t5[1291] := -0.0266525;
   t5[1292] := -0.0273713;
   t5[1293] := -0.0280848;
   t5[1294] := -0.0287929;
   t5[1295] := -0.0294957;
   t5[1296] := -0.0301934;
   t5[1297] := -0.030886;
   t5[1298] := -0.0315736;
   t5[1299] := -0.0322563;
   t5[1300] := 0.1115208;
   t5[1301] := 0.1124736;
   t5[1302] := 0.113418;
   t5[1303] := 0.1143538;
   t5[1304] := 0.1152811;
   t5[1305] := 0.1161997;
   t5[1306] := 0.1171098;
   t5[1307] := 0.1180112;
   t5[1308] := 0.1189039;
   t5[1309] := 0.1197878;
   t5[1310] := 0.120663;
   t5[1311] := 0.1215294;
   t5[1312] := 0.1223869;
   t5[1313] := 0.1232356;
   t5[1314] := 0.1240754;
   t5[1315] := 0.1249062;
   t5[1316] := 0.125728;
   t5[1317] := 0.1265409;
   t5[1318] := 0.1273447;
   t5[1319] := 0.1281394;
   t5[1320] := 0.128925;
   t5[1321] := 0.1297014;
   t5[1322] := 0.1304687;
   t5[1323] := 0.1312267;
   t5[1324] := 0.1319755;
   t5[1325] := 0.132715;
   t5[1326] := 0.1334452;
   t5[1327] := 0.134166;
   t5[1328] := 0.1348774;
   t5[1329] := 0.1355794;
   t5[1330] := 0.1362719;
   t5[1331] := 0.136955;
   t5[1332] := 0.1376285;
   t5[1333] := 0.1382924;
   t5[1334] := 0.1389468;
   t5[1335] := 0.1395914;
   t5[1336] := 0.1402262;
   t5[1337] := 0.140851;
   t5[1338] := 0.1414657;
   t5[1339] := 0.1420702;
   t5[1340] := 0.1426643;
   t5[1341] := 0.1432479;
   t5[1342] := 0.1438208;
   t5[1343] := 0.144383;
   t5[1344] := 0.1449343;
   t5[1345] := 0.1454746;
   t5[1346] := 0.1460037;
   t5[1347] := 0.1465215;
   t5[1348] := 0.1470279;
   t5[1349] := 0.1475227;
   t5[1350] := 0.0927025;
   t5[1351] := 0.0930827;
   t5[1352] := 0.0934529;
   t5[1353] := 0.0938132;
   t5[1354] := 0.0941636;
   t5[1355] := 0.094504;
   t5[1356] := 0.0948345;
   t5[1357] := 0.0951551;
   t5[1358] := 0.0954658;
   t5[1359] := 0.0957665;
   t5[1360] := 0.0960574;
   t5[1361] := 0.0963383;
   t5[1362] := 0.0966094;
   t5[1363] := 0.0968706;
   t5[1364] := 0.0971219;
   t5[1365] := 0.0973634;
   t5[1366] := 0.097595;
   t5[1367] := 0.0978168;
   t5[1368] := 0.0980287;
   t5[1369] := 0.0982308;
   t5[1370] := 0.098423;
   t5[1371] := 0.0986054;
   t5[1372] := 0.0987781;
   t5[1373] := 0.0989409;
   t5[1374] := 0.0990939;
   t5[1375] := 0.0992371;
   t5[1376] := 0.0993705;
   t5[1377] := 0.0994942;
   t5[1378] := 0.0996081;
   t5[1379] := 0.0997122;
   t5[1380] := 0.0998065;
   t5[1381] := 0.0998911;
   t5[1382] := 0.099966;
   t5[1383] := 0.1000311;
   t5[1384] := 0.1000866;
   t5[1385] := 0.1001323;
   t5[1386] := 0.1001685;
   t5[1387] := 0.1001953;
   t5[1388] := 0.1002128;
   t5[1389] := 0.100221;
   t5[1390] := 0.1002201;
   t5[1391] := 0.1002102;
   t5[1392] := 0.1001915;
   t5[1393] := 0.1001639;
   t5[1394] := 0.1001276;
   t5[1395] := 0.1000828;
   t5[1396] := 0.1000295;
   t5[1397] := 0.0999678;
   t5[1398] := 0.0998978;
   t5[1399] := 0.0998198;
   t5[1400] := 0.1446864;
   t5[1401] := 0.1450943;
   t5[1402] := 0.1454921;
   t5[1403] := 0.1458796;
   t5[1404] := 0.1462567;
   t5[1405] := 0.1466235;
   t5[1406] := 0.1469798;
   t5[1407] := 0.1473257;
   t5[1408] := 0.1476611;
   t5[1409] := 0.1479859;
   t5[1410] := 0.1483001;
   t5[1411] := 0.1486036;
   t5[1412] := 0.1488965;
   t5[1413] := 0.1491785;
   t5[1414] := 0.1494499;
   t5[1415] := 0.1497103;
   t5[1416] := 0.1499599;
   t5[1417] := 0.1501985;
   t5[1418] := 0.1504261;
   t5[1419] := 0.1506428;
   t5[1420] := 0.1508483;
   t5[1421] := 0.1510427;
   t5[1422] := 0.151226;
   t5[1423] := 0.151398;
   t5[1424] := 0.1515587;
   t5[1425] := 0.1517082;
   t5[1426] := 0.1518463;
   t5[1427] := 0.1519729;
   t5[1428] := 0.1520882;
   t5[1429] := 0.1521919;
   t5[1430] := 0.1522841;
   t5[1431] := 0.1523647;
   t5[1432] := 0.1524337;
   t5[1433] := 0.1524909;
   t5[1434] := 0.1525365;
   t5[1435] := 0.1525704;
   t5[1436] := 0.1525928;
   t5[1437] := 0.1526038;
   t5[1438] := 0.1526037;
   t5[1439] := 0.1525925;
   t5[1440] := 0.1525703;
   t5[1441] := 0.1525374;
   t5[1442] := 0.1524938;
   t5[1443] := 0.1524398;
   t5[1444] := 0.1523754;
   t5[1445] := 0.1523009;
   t5[1446] := 0.1522162;
   t5[1447] := 0.1521217;
   t5[1448] := 0.1520174;
   t5[1449] := 0.1519035;
   t5[1450] := -0.0403738;
   t5[1451] := -0.0395231;
   t5[1452] := -0.0386606;
   t5[1453] := -0.0377861;
   t5[1454] := -0.0368996;
   t5[1455] := -0.0360007;
   t5[1456] := -0.0350893;
   t5[1457] := -0.0341651;
   t5[1458] := -0.0332281;
   t5[1459] := -0.0322779;
   t5[1460] := -0.0313144;
   t5[1461] := -0.0303373;
   t5[1462] := -0.0293466;
   t5[1463] := -0.028342;
   t5[1464] := -0.0273232;
   t5[1465] := -0.0262901;
   t5[1466] := -0.0252426;
   t5[1467] := -0.0241803;
   t5[1468] := -0.0231032;
   t5[1469] := -0.022011;
   t5[1470] := -0.0209035;
   t5[1471] := -0.0197805;
   t5[1472] := -0.0186418;
   t5[1473] := -0.0174872;
   t5[1474] := -0.0163166;
   t5[1475] := -0.0151297;
   t5[1476] := -0.0139263;
   t5[1477] := -0.0127063;
   t5[1478] := -0.0114694;
   t5[1479] := -0.0102154;
   t5[1480] := -0.0089442;
   t5[1481] := -0.0076555;
   t5[1482] := -0.0063492;
   t5[1483] := -0.005025;
   t5[1484] := -0.0036829;
   t5[1485] := -0.0023229;
   t5[1486] := -0.0009455;
   t5[1487] := 0.0004488;
   t5[1488] := 0.0018596;
   t5[1489] := 0.0032865;
   t5[1490] := 0.0047291;
   t5[1491] := 0.0061869;
   t5[1492] := 0.0076596;
   t5[1493] := 0.0091467;
   t5[1494] := 0.0106478;
   t5[1495] := 0.0121624;
   t5[1496] := 0.0136901;
   t5[1497] := 0.0152306;
   t5[1498] := 0.0167833;
   t5[1499] := 0.018348;
   t5[1500] := 0.1207302;
   t5[1501] := 0.1212353;
   t5[1502] := 0.1217364;
   t5[1503] := 0.1222335;
   t5[1504] := 0.1227265;
   t5[1505] := 0.1232155;
   t5[1506] := 0.1237005;
   t5[1507] := 0.1241813;
   t5[1508] := 0.1246581;
   t5[1509] := 0.1251307;
   t5[1510] := 0.1255992;
   t5[1511] := 0.1260636;
   t5[1512] := 0.1265237;
   t5[1513] := 0.1269798;
   t5[1514] := 0.1274316;
   t5[1515] := 0.1278793;
   t5[1516] := 0.1283227;
   t5[1517] := 0.1287618;
   t5[1518] := 0.1291968;
   t5[1519] := 0.1296274;
   t5[1520] := 0.1300538;
   t5[1521] := 0.1304759;
   t5[1522] := 0.1308936;
   t5[1523] := 0.1313071;
   t5[1524] := 0.1317161;
   t5[1525] := 0.1321208;
   t5[1526] := 0.1325212;
   t5[1527] := 0.1329171;
   t5[1528] := 0.1333087;
   t5[1529] := 0.1336958;
   t5[1530] := 0.1340785;
   t5[1531] := 0.1344567;
   t5[1532] := 0.1348305;
   t5[1533] := 0.1351997;
   t5[1534] := 0.1355645;
   t5[1535] := 0.1359247;
   t5[1536] := 0.1362803;
   t5[1537] := 0.1366311;
   t5[1538] := 0.1369772;
   t5[1539] := 0.1373184;
   t5[1540] := 0.1376546;
   t5[1541] := 0.1379859;
   t5[1542] := 0.138312;
   t5[1543] := 0.138633;
   t5[1544] := 0.1389486;
   t5[1545] := 0.139259;
   t5[1546] := 0.139564;
   t5[1547] := 0.1398635;
   t5[1548] := 0.1401574;
   t5[1549] := 0.1404457;
   t5[1550] := 0.2641891;
   t5[1551] := 0.261912;
   t5[1552] := 0.2596165;
   t5[1553] := 0.2573028;
   t5[1554] := 0.2549714;
   t5[1555] := 0.2526227;
   t5[1556] := 0.250257;
   t5[1557] := 0.2478748;
   t5[1558] := 0.2454765;
   t5[1559] := 0.2430624;
   t5[1560] := 0.240633;
   t5[1561] := 0.2381887;
   t5[1562] := 0.2357297;
   t5[1563] := 0.2332567;
   t5[1564] := 0.2307699;
   t5[1565] := 0.2282697;
   t5[1566] := 0.2257565;
   t5[1567] := 0.2232308;
   t5[1568] := 0.2206929;
   t5[1569] := 0.2181432;
   t5[1570] := 0.2155821;
   t5[1571] := 0.2130101;
   t5[1572] := 0.2104274;
   t5[1573] := 0.2078346;
   t5[1574] := 0.2052319;
   t5[1575] := 0.2026199;
   t5[1576] := 0.1999989;
   t5[1577] := 0.1973692;
   t5[1578] := 0.1947314;
   t5[1579] := 0.1920857;
   t5[1580] := 0.1894325;
   t5[1581] := 0.1867724;
   t5[1582] := 0.1841056;
   t5[1583] := 0.1814327;
   t5[1584] := 0.1787538;
   t5[1585] := 0.1760694;
   t5[1586] := 0.1733797;
   t5[1587] := 0.1706849;
   t5[1588] := 0.1679854;
   t5[1589] := 0.1652812;
   t5[1590] := 0.1625728;
   t5[1591] := 0.1598602;
   t5[1592] := 0.1571439;
   t5[1593] := 0.154424;
   t5[1594] := 0.1517007;
   t5[1595] := 0.1489744;
   t5[1596] := 0.1462451;
   t5[1597] := 0.1435134;
   t5[1598] := 0.1407792;
   t5[1599] := 0.138043;
   t5[1600] := -0.013076;
   t5[1601] := -0.0118497;
   t5[1602] := -0.0106312;
   t5[1603] := -0.0094206;
   t5[1604] := -0.0082182;
   t5[1605] := -0.0070242;
   t5[1606] := -0.0058388;
   t5[1607] := -0.0046621;
   t5[1608] := -0.0034945;
   t5[1609] := -0.0023362;
   t5[1610] := -0.0011873;
   t5[1611] := -4.81E-05;
   t5[1612] := 0.0010812;
   t5[1613] := 0.0022004;
   t5[1614] := 0.0033093;
   t5[1615] := 0.0044077;
   t5[1616] := 0.0054953;
   t5[1617] := 0.0065719;
   t5[1618] := 0.0076374;
   t5[1619] := 0.0086914;
   t5[1620] := 0.0097339;
   t5[1621] := 0.0107645;
   t5[1622] := 0.0117831;
   t5[1623] := 0.0127894;
   t5[1624] := 0.0137832;
   t5[1625] := 0.0147644;
   t5[1626] := 0.0157326;
   t5[1627] := 0.0166878;
   t5[1628] := 0.0176295;
   t5[1629] := 0.0185578;
   t5[1630] := 0.0194723;
   t5[1631] := 0.0203728;
   t5[1632] := 0.0212591;
   t5[1633] := 0.022131;
   t5[1634] := 0.0229882;
   t5[1635] := 0.023831;
   t5[1636] := 0.0246595;
   t5[1637] := 0.0254739;
   t5[1638] := 0.0262744;
   t5[1639] := 0.0270614;
   t5[1640] := 0.0278349;
   t5[1641] := 0.0285953;
   t5[1642] := 0.0293428;
   t5[1643] := 0.0300776;
   t5[1644] := 0.0307999;
   t5[1645] := 0.0315099;
   t5[1646] := 0.0322079;
   t5[1647] := 0.0328942;
   t5[1648] := 0.0335689;
   t5[1649] := 0.0342322;
   t5[1650] := -0.0208986;
   t5[1651] := -0.0213763;
   t5[1652] := -0.021847;
   t5[1653] := -0.0223105;
   t5[1654] := -0.0227665;
   t5[1655] := -0.0232147;
   t5[1656] := -0.0236548;
   t5[1657] := -0.0240864;
   t5[1658] := -0.0245092;
   t5[1659] := -0.024923;
   t5[1660] := -0.0253275;
   t5[1661] := -0.0257222;
   t5[1662] := -0.026107;
   t5[1663] := -0.0264815;
   t5[1664] := -0.0268454;
   t5[1665] := -0.0271984;
   t5[1666] := -0.0275402;
   t5[1667] := -0.0278705;
   t5[1668] := -0.028189;
   t5[1669] := -0.0284953;
   t5[1670] := -0.0287892;
   t5[1671] := -0.0290703;
   t5[1672] := -0.0293384;
   t5[1673] := -0.0295931;
   t5[1674] := -0.0298342;
   t5[1675] := -0.0300612;
   t5[1676] := -0.030274;
   t5[1677] := -0.0304722;
   t5[1678] := -0.0306555;
   t5[1679] := -0.0308236;
   t5[1680] := -0.0309761;
   t5[1681] := -0.0311129;
   t5[1682] := -0.0312335;
   t5[1683] := -0.0313376;
   t5[1684] := -0.0314251;
   t5[1685] := -0.0314958;
   t5[1686] := -0.03155;
   t5[1687] := -0.0315877;
   t5[1688] := -0.0316091;
   t5[1689] := -0.0316144;
   t5[1690] := -0.0316038;
   t5[1691] := -0.0315773;
   t5[1692] := -0.0315351;
   t5[1693] := -0.0314774;
   t5[1694] := -0.0314044;
   t5[1695] := -0.0313161;
   t5[1696] := -0.0312127;
   t5[1697] := -0.0310944;
   t5[1698] := -0.0309614;
   t5[1699] := -0.0308137;
   t5[1700] := -0.0136591;
   t5[1701] := -0.0132589;
   t5[1702] := -0.0128679;
   t5[1703] := -0.0124862;
   t5[1704] := -0.012114;
   t5[1705] := -0.0117512;
   t5[1706] := -0.0113981;
   t5[1707] := -0.0110547;
   t5[1708] := -0.010721;
   t5[1709] := -0.0103972;
   t5[1710] := -0.0100834;
   t5[1711] := -0.0097797;
   t5[1712] := -0.0094861;
   t5[1713] := -0.0092027;
   t5[1714] := -0.0089297;
   t5[1715] := -0.0086671;
   t5[1716] := -0.008415;
   t5[1717] := -0.0081735;
   t5[1718] := -0.0079427;
   t5[1719] := -0.0077228;
   t5[1720] := -0.0075137;
   t5[1721] := -0.0073155;
   t5[1722] := -0.0071285;
   t5[1723] := -0.0069526;
   t5[1724] := -0.0067879;
   t5[1725] := -0.0066346;
   t5[1726] := -0.0064928;
   t5[1727] := -0.0063624;
   t5[1728] := -0.0062437;
   t5[1729] := -0.0061367;
   t5[1730] := -0.0060414;
   t5[1731] := -0.0059581;
   t5[1732] := -0.0058867;
   t5[1733] := -0.0058275;
   t5[1734] := -0.0057803;
   t5[1735] := -0.0057453;
   t5[1736] := -0.0057221;
   t5[1737] := -0.0057108;
   t5[1738] := -0.005711;
   t5[1739] := -0.0057226;
   t5[1740] := -0.0057455;
   t5[1741] := -0.0057796;
   t5[1742] := -0.0058246;
   t5[1743] := -0.0058803;
   t5[1744] := -0.0059467;
   t5[1745] := -0.0060236;
   t5[1746] := -0.0061108;
   t5[1747] := -0.0062082;
   t5[1748] := -0.0063155;
   t5[1749] := -0.0064327;
   t5[1750] := -0.014299;
   t5[1751] := -0.0131987;
   t5[1752] := -0.012092;
   t5[1753] := -0.0109787;
   t5[1754] := -0.0098588;
   t5[1755] := -0.0087325;
   t5[1756] := -0.0075996;
   t5[1757] := -0.0064601;
   t5[1758] := -0.005314;
   t5[1759] := -0.0041614;
   t5[1760] := -0.0030022;
   t5[1761] := -0.0018365;
   t5[1762] := -0.0006641;
   t5[1763] := 0.0005149;
   t5[1764] := 0.0017005;
   t5[1765] := 0.0028927;
   t5[1766] := 0.0040916;
   t5[1767] := 0.0052971;
   t5[1768] := 0.0065092;
   t5[1769] := 0.007728;
   t5[1770] := 0.0089534;
   t5[1771] := 0.0101856;
   t5[1772] := 0.0114244;
   t5[1773] := 0.0126699;
   t5[1774] := 0.013922;
   t5[1775] := 0.0151809;
   t5[1776] := 0.0164465;
   t5[1777] := 0.0177188;
   t5[1778] := 0.0189979;
   t5[1779] := 0.0202837;
   t5[1780] := 0.0215762;
   t5[1781] := 0.0228755;
   t5[1782] := 0.0241815;
   t5[1783] := 0.0254943;
   t5[1784] := 0.0268139;
   t5[1785] := 0.0281401;
   t5[1786] := 0.0294727;
   t5[1787] := 0.0308115;
   t5[1788] := 0.0321562;
   t5[1789] := 0.0335066;
   t5[1790] := 0.0348626;
   t5[1791] := 0.0362239;
   t5[1792] := 0.0375902;
   t5[1793] := 0.0389613;
   t5[1794] := 0.0403371;
   t5[1795] := 0.0417173;
   t5[1796] := 0.0431016;
   t5[1797] := 0.0444899;
   t5[1798] := 0.045882;
   t5[1799] := 0.0472775;
   t5[1800] := -0.0809446;
   t5[1801] := -0.0811497;
   t5[1802] := -0.0813545;
   t5[1803] := -0.0815591;
   t5[1804] := -0.0817636;
   t5[1805] := -0.0819682;
   t5[1806] := -0.0821731;
   t5[1807] := -0.0823782;
   t5[1808] := -0.0825839;
   t5[1809] := -0.08279;
   t5[1810] := -0.0829969;
   t5[1811] := -0.0832046;
   t5[1812] := -0.0834133;
   t5[1813] := -0.083623;
   t5[1814] := -0.0838339;
   t5[1815] := -0.0840461;
   t5[1816] := -0.0842598;
   t5[1817] := -0.084475;
   t5[1818] := -0.084692;
   t5[1819] := -0.0849107;
   t5[1820] := -0.0851314;
   t5[1821] := -0.0853541;
   t5[1822] := -0.0855791;
   t5[1823] := -0.0858063;
   t5[1824] := -0.086036;
   t5[1825] := -0.0862682;
   t5[1826] := -0.0865031;
   t5[1827] := -0.0867409;
   t5[1828] := -0.0869815;
   t5[1829] := -0.0872252;
   t5[1830] := -0.0874721;
   t5[1831] := -0.0877223;
   t5[1832] := -0.0879759;
   t5[1833] := -0.0882331;
   t5[1834] := -0.0884939;
   t5[1835] := -0.0887583;
   t5[1836] := -0.0890261;
   t5[1837] := -0.0892972;
   t5[1838] := -0.0895712;
   t5[1839] := -0.0898482;
   t5[1840] := -0.0901278;
   t5[1841] := -0.09041;
   t5[1842] := -0.0906944;
   t5[1843] := -0.0909811;
   t5[1844] := -0.0912697;
   t5[1845] := -0.0915601;
   t5[1846] := -0.0918521;
   t5[1847] := -0.0921455;
   t5[1848] := -0.0924402;
   t5[1849] := -0.092736;
   t5[1850] := 0.0001257;
   t5[1851] := 0.0009313;
   t5[1852] := 0.0017379;
   t5[1853] := 0.0025455;
   t5[1854] := 0.0033542;
   t5[1855] := 0.004164;
   t5[1856] := 0.0049749;
   t5[1857] := 0.0057871;
   t5[1858] := 0.0066004;
   t5[1859] := 0.0074149;
   t5[1860] := 0.0082308;
   t5[1861] := 0.009048;
   t5[1862] := 0.0098665;
   t5[1863] := 0.0106864;
   t5[1864] := 0.0115078;
   t5[1865] := 0.0123306;
   t5[1866] := 0.0131549;
   t5[1867] := 0.0139808;
   t5[1868] := 0.0148082;
   t5[1869] := 0.0156372;
   t5[1870] := 0.0164679;
   t5[1871] := 0.0173003;
   t5[1872] := 0.0181343;
   t5[1873] := 0.0189702;
   t5[1874] := 0.0198078;
   t5[1875] := 0.0206472;
   t5[1876] := 0.0214885;
   t5[1877] := 0.0223317;
   t5[1878] := 0.0231768;
   t5[1879] := 0.0240239;
   t5[1880] := 0.024873;
   t5[1881] := 0.0257241;
   t5[1882] := 0.0265774;
   t5[1883] := 0.0274327;
   t5[1884] := 0.0282902;
   t5[1885] := 0.0291498;
   t5[1886] := 0.0300117;
   t5[1887] := 0.030876;
   t5[1888] := 0.0317425;
   t5[1889] := 0.0326115;
   t5[1890] := 0.0334829;
   t5[1891] := 0.0343568;
   t5[1892] := 0.0352333;
   t5[1893] := 0.0361124;
   t5[1894] := 0.0369941;
   t5[1895] := 0.0378785;
   t5[1896] := 0.0387658;
   t5[1897] := 0.0396558;
   t5[1898] := 0.0405487;
   t5[1899] := 0.0414445;
   t5[1900] := -0.0673197;
   t5[1901] := -0.0672477;
   t5[1902] := -0.0671676;
   t5[1903] := -0.0670793;
   t5[1904] := -0.0669828;
   t5[1905] := -0.066878;
   t5[1906] := -0.0667649;
   t5[1907] := -0.0666434;
   t5[1908] := -0.0665134;
   t5[1909] := -0.066375;
   t5[1910] := -0.0662281;
   t5[1911] := -0.0660726;
   t5[1912] := -0.0659084;
   t5[1913] := -0.0657357;
   t5[1914] := -0.0655542;
   t5[1915] := -0.0653639;
   t5[1916] := -0.0651649;
   t5[1917] := -0.0649569;
   t5[1918] := -0.0647401;
   t5[1919] := -0.0645144;
   t5[1920] := -0.0642796;
   t5[1921] := -0.0640358;
   t5[1922] := -0.0637829;
   t5[1923] := -0.0635209;
   t5[1924] := -0.0632497;
   t5[1925] := -0.0629693;
   t5[1926] := -0.0626796;
   t5[1927] := -0.0623805;
   t5[1928] := -0.0620721;
   t5[1929] := -0.0617543;
   t5[1930] := -0.061427;
   t5[1931] := -0.0610902;
   t5[1932] := -0.0607438;
   t5[1933] := -0.0603878;
   t5[1934] := -0.0600222;
   t5[1935] := -0.0596471;
   t5[1936] := -0.0592627;
   t5[1937] := -0.0588692;
   t5[1938] := -0.0584668;
   t5[1939] := -0.0580558;
   t5[1940] := -0.0576364;
   t5[1941] := -0.0572089;
   t5[1942] := -0.0567733;
   t5[1943] := -0.05633;
   t5[1944] := -0.0558792;
   t5[1945] := -0.0554211;
   t5[1946] := -0.0549559;
   t5[1947] := -0.0544838;
   t5[1948] := -0.0540051;
   t5[1949] := -0.05352;
   t5[1950] := 0.0792828;
   t5[1951] := 0.0784182;
   t5[1952] := 0.0775534;
   t5[1953] := 0.0766885;
   t5[1954] := 0.0758237;
   t5[1955] := 0.0749592;
   t5[1956] := 0.0740953;
   t5[1957] := 0.073232;
   t5[1958] := 0.0723696;
   t5[1959] := 0.0715082;
   t5[1960] := 0.0706481;
   t5[1961] := 0.0697895;
   t5[1962] := 0.0689324;
   t5[1963] := 0.0680772;
   t5[1964] := 0.067224;
   t5[1965] := 0.066373;
   t5[1966] := 0.0655243;
   t5[1967] := 0.0646782;
   t5[1968] := 0.0638348;
   t5[1969] := 0.0629944;
   t5[1970] := 0.0621571;
   t5[1971] := 0.0613231;
   t5[1972] := 0.0604927;
   t5[1973] := 0.0596659;
   t5[1974] := 0.0588429;
   t5[1975] := 0.0580241;
   t5[1976] := 0.0572094;
   t5[1977] := 0.0563992;
   t5[1978] := 0.0555937;
   t5[1979] := 0.0547929;
   t5[1980] := 0.0539971;
   t5[1981] := 0.0532065;
   t5[1982] := 0.0524213;
   t5[1983] := 0.0516417;
   t5[1984] := 0.0508677;
   t5[1985] := 0.0500996;
   t5[1986] := 0.0493373;
   t5[1987] := 0.0485808;
   t5[1988] := 0.0478301;
   t5[1989] := 0.0470852;
   t5[1990] := 0.0463462;
   t5[1991] := 0.045613;
   t5[1992] := 0.0448857;
   t5[1993] := 0.0441641;
   t5[1994] := 0.0434485;
   t5[1995] := 0.0427387;
   t5[1996] := 0.0420348;
   t5[1997] := 0.0413367;
   t5[1998] := 0.0406445;
   t5[1999] := 0.0399582;
   t5[2000] := -0.1993882;
   t5[2001] := -0.1987197;
   t5[2002] := -0.1980445;
   t5[2003] := -0.1973628;
   t5[2004] := -0.1966745;
   t5[2005] := -0.1959796;
   t5[2006] := -0.1952783;
   t5[2007] := -0.1945705;
   t5[2008] := -0.1938564;
   t5[2009] := -0.1931358;
   t5[2010] := -0.192409;
   t5[2011] := -0.1916759;
   t5[2012] := -0.1909366;
   t5[2013] := -0.1901912;
   t5[2014] := -0.1894396;
   t5[2015] := -0.1886819;
   t5[2016] := -0.1879182;
   t5[2017] := -0.1871485;
   t5[2018] := -0.1863728;
   t5[2019] := -0.1855913;
   t5[2020] := -0.1848039;
   t5[2021] := -0.1840106;
   t5[2022] := -0.1832116;
   t5[2023] := -0.1824069;
   t5[2024] := -0.1815965;
   t5[2025] := -0.1807804;
   t5[2026] := -0.1799588;
   t5[2027] := -0.1791316;
   t5[2028] := -0.1782989;
   t5[2029] := -0.1774607;
   t5[2030] := -0.1766172;
   t5[2031] := -0.1757682;
   t5[2032] := -0.174914;
   t5[2033] := -0.1740544;
   t5[2034] := -0.1731896;
   t5[2035] := -0.1723197;
   t5[2036] := -0.1714448;
   t5[2037] := -0.1705651;
   t5[2038] := -0.1696807;
   t5[2039] := -0.1687917;
   t5[2040] := -0.1678983;
   t5[2041] := -0.1670006;
   t5[2042] := -0.1660989;
   t5[2043] := -0.1651931;
   t5[2044] := -0.1642835;
   t5[2045] := -0.1633702;
   t5[2046] := -0.1624534;
   t5[2047] := -0.1615331;
   t5[2048] := -0.1606096;
   t5[2049] := -0.159683;
   t5[2050] := -0.110986;
   t5[2051] := -0.1115587;
   t5[2052] := -0.1121124;
   t5[2053] := -0.1126469;
   t5[2054] := -0.1131621;
   t5[2055] := -0.1136579;
   t5[2056] := -0.114134;
   t5[2057] := -0.1145904;
   t5[2058] := -0.1150269;
   t5[2059] := -0.1154433;
   t5[2060] := -0.1158395;
   t5[2061] := -0.1162154;
   t5[2062] := -0.1165708;
   t5[2063] := -0.1169056;
   t5[2064] := -0.1172196;
   t5[2065] := -0.1175127;
   t5[2066] := -0.1177848;
   t5[2067] := -0.1180356;
   t5[2068] := -0.118265;
   t5[2069] := -0.118473;
   t5[2070] := -0.1186593;
   t5[2071] := -0.1188239;
   t5[2072] := -0.1189664;
   t5[2073] := -0.119087;
   t5[2074] := -0.1191852;
   t5[2075] := -0.1192611;
   t5[2076] := -0.1193145;
   t5[2077] := -0.1193452;
   t5[2078] := -0.1193531;
   t5[2079] := -0.1193381;
   t5[2080] := -0.1192999;
   t5[2081] := -0.1192385;
   t5[2082] := -0.1191538;
   t5[2083] := -0.1190454;
   t5[2084] := -0.1189135;
   t5[2085] := -0.1187581;
   t5[2086] := -0.1185796;
   t5[2087] := -0.1183784;
   t5[2088] := -0.1181548;
   t5[2089] := -0.1179094;
   t5[2090] := -0.1176424;
   t5[2091] := -0.1173542;
   t5[2092] := -0.1170453;
   t5[2093] := -0.1167159;
   t5[2094] := -0.1163665;
   t5[2095] := -0.1159974;
   t5[2096] := -0.1156091;
   t5[2097] := -0.1152018;
   t5[2098] := -0.114776;
   t5[2099] := -0.1143322;
   t5[2100] := -0.0163093;
   t5[2101] := -0.0173279;
   t5[2102] := -0.0183363;
   t5[2103] := -0.0193342;
   t5[2104] := -0.0203215;
   t5[2105] := -0.0212978;
   t5[2106] := -0.0222629;
   t5[2107] := -0.0232166;
   t5[2108] := -0.0241586;
   t5[2109] := -0.0250886;
   t5[2110] := -0.0260066;
   t5[2111] := -0.0269121;
   t5[2112] := -0.027805;
   t5[2113] := -0.0286849;
   t5[2114] := -0.0295518;
   t5[2115] := -0.0304053;
   t5[2116] := -0.0312451;
   t5[2117] := -0.0320711;
   t5[2118] := -0.0328829;
   t5[2119] := -0.0336804;
   t5[2120] := -0.0344633;
   t5[2121] := -0.0352314;
   t5[2122] := -0.0359844;
   t5[2123] := -0.036722;
   t5[2124] := -0.0374441;
   t5[2125] := -0.0381503;
   t5[2126] := -0.0388405;
   t5[2127] := -0.0395144;
   t5[2128] := -0.0401717;
   t5[2129] := -0.0408123;
   t5[2130] := -0.0414358;
   t5[2131] := -0.042042;
   t5[2132] := -0.0426307;
   t5[2133] := -0.0432016;
   t5[2134] := -0.0437546;
   t5[2135] := -0.0442896;
   t5[2136] := -0.0448069;
   t5[2137] := -0.0453067;
   t5[2138] := -0.0457891;
   t5[2139] := -0.0462545;
   t5[2140] := -0.046703;
   t5[2141] := -0.0471348;
   t5[2142] := -0.0475501;
   t5[2143] := -0.0479492;
   t5[2144] := -0.0483322;
   t5[2145] := -0.0486994;
   t5[2146] := -0.049051;
   t5[2147] := -0.0493871;
   t5[2148] := -0.049708;
   t5[2149] := -0.0500139;
   t5[2150] := 0.0848828;
   t5[2151] := 0.0840354;
   t5[2152] := 0.0831941;
   t5[2153] := 0.0823589;
   t5[2154] := 0.0815301;
   t5[2155] := 0.080708;
   t5[2156] := 0.0798927;
   t5[2157] := 0.0790844;
   t5[2158] := 0.0782833;
   t5[2159] := 0.0774897;
   t5[2160] := 0.0767036;
   t5[2161] := 0.0759254;
   t5[2162] := 0.0751553;
   t5[2163] := 0.0743934;
   t5[2164] := 0.0736399;
   t5[2165] := 0.072895;
   t5[2166] := 0.072159;
   t5[2167] := 0.0714321;
   t5[2168] := 0.0707144;
   t5[2169] := 0.0700061;
   t5[2170] := 0.0693075;
   t5[2171] := 0.0686188;
   t5[2172] := 0.0679401;
   t5[2173] := 0.0672716;
   t5[2174] := 0.0666136;
   t5[2175] := 0.0659663;
   t5[2176] := 0.0653299;
   t5[2177] := 0.0647045;
   t5[2178] := 0.0640904;
   t5[2179] := 0.0634877;
   t5[2180] := 0.0628968;
   t5[2181] := 0.0623177;
   t5[2182] := 0.0617507;
   t5[2183] := 0.0611959;
   t5[2184] := 0.0606536;
   t5[2185] := 0.0601237;
   t5[2186] := 0.0596059;
   t5[2187] := 0.0591;
   t5[2188] := 0.0586057;
   t5[2189] := 0.0581228;
   t5[2190] := 0.0576511;
   t5[2191] := 0.0571902;
   t5[2192] := 0.05674;
   t5[2193] := 0.0563001;
   t5[2194] := 0.0558704;
   t5[2195] := 0.0554507;
   t5[2196] := 0.0550406;
   t5[2197] := 0.0546399;
   t5[2198] := 0.0542484;
   t5[2199] := 0.0538658;
   t5[2200] := -0.0819279;
   t5[2201] := -0.0824729;
   t5[2202] := -0.0830032;
   t5[2203] := -0.083518;
   t5[2204] := -0.0840171;
   t5[2205] := -0.0844999;
   t5[2206] := -0.0849661;
   t5[2207] := -0.085415;
   t5[2208] := -0.0858463;
   t5[2209] := -0.0862595;
   t5[2210] := -0.0866541;
   t5[2211] := -0.0870298;
   t5[2212] := -0.0873859;
   t5[2213] := -0.0877222;
   t5[2214] := -0.088038;
   t5[2215] := -0.0883331;
   t5[2216] := -0.0886068;
   t5[2217] := -0.0888587;
   t5[2218] := -0.0890884;
   t5[2219] := -0.0892954;
   t5[2220] := -0.0894793;
   t5[2221] := -0.0896396;
   t5[2222] := -0.0897759;
   t5[2223] := -0.0898876;
   t5[2224] := -0.0899743;
   t5[2225] := -0.0900356;
   t5[2226] := -0.090071;
   t5[2227] := -0.09008;
   t5[2228] := -0.0900622;
   t5[2229] := -0.0900172;
   t5[2230] := -0.0899444;
   t5[2231] := -0.0898434;
   t5[2232] := -0.0897138;
   t5[2233] := -0.0895551;
   t5[2234] := -0.0893668;
   t5[2235] := -0.0891493;
   t5[2236] := -0.0889028;
   t5[2237] := -0.088628;
   t5[2238] := -0.0883254;
   t5[2239] := -0.0879954;
   t5[2240] := -0.0876385;
   t5[2241] := -0.0872553;
   t5[2242] := -0.0868462;
   t5[2243] := -0.0864116;
   t5[2244] := -0.0859523;
   t5[2245] := -0.0854685;
   t5[2246] := -0.0849609;
   t5[2247] := -0.0844299;
   t5[2248] := -0.0838759;
   t5[2249] := -0.0832996;
   t5[2250] := -0.0222091;
   t5[2251] := -0.0213377;
   t5[2252] := -0.0204763;
   t5[2253] := -0.0196253;
   t5[2254] := -0.0187854;
   t5[2255] := -0.017957;
   t5[2256] := -0.0171404;
   t5[2257] := -0.0163363;
   t5[2258] := -0.0155452;
   t5[2259] := -0.0147674;
   t5[2260] := -0.0140035;
   t5[2261] := -0.013254;
   t5[2262] := -0.0125193;
   t5[2263] := -0.0118;
   t5[2264] := -0.0110964;
   t5[2265] := -0.0104092;
   t5[2266] := -0.0097388;
   t5[2267] := -0.0090856;
   t5[2268] := -0.0084502;
   t5[2269] := -0.007833;
   t5[2270] := -0.0072345;
   t5[2271] := -0.0066552;
   t5[2272] := -0.0060956;
   t5[2273] := -0.0055562;
   t5[2274] := -0.0050374;
   t5[2275] := -0.0045398;
   t5[2276] := -0.0040638;
   t5[2277] := -0.0036099;
   t5[2278] := -0.0031786;
   t5[2279] := -0.0027703;
   t5[2280] := -0.0023856;
   t5[2281] := -0.002025;
   t5[2282] := -0.0016888;
   t5[2283] := -0.0013777;
   t5[2284] := -0.001092;
   t5[2285] := -0.0008317;
   t5[2286] := -0.0005967;
   t5[2287] := -0.0003866;
   t5[2288] := -0.0002013;
   t5[2289] := -4.04E-05;
   t5[2290] := 9.62E-05;
   t5[2291] := 0.0002089;
   t5[2292] := 0.0002977;
   t5[2293] := 0.0003631;
   t5[2294] := 0.0004053;
   t5[2295] := 0.0004244;
   t5[2296] := 0.0004207;
   t5[2297] := 0.0003945;
   t5[2298] := 0.000346;
   t5[2299] := 0.0002755;
   t5[2300] := -0.0469918;
   t5[2301] := -0.0460147;
   t5[2302] := -0.045055;
   t5[2303] := -0.0441128;
   t5[2304] := -0.0431885;
   t5[2305] := -0.0422822;
   t5[2306] := -0.0413941;
   t5[2307] := -0.0405246;
   t5[2308] := -0.0396739;
   t5[2309] := -0.0388421;
   t5[2310] := -0.0380297;
   t5[2311] := -0.0372368;
   t5[2312] := -0.0364636;
   t5[2313] := -0.0357104;
   t5[2314] := -0.0349775;
   t5[2315] := -0.034265;
   t5[2316] := -0.0335733;
   t5[2317] := -0.0329026;
   t5[2318] := -0.0322531;
   t5[2319] := -0.0316251;
   t5[2320] := -0.0310187;
   t5[2321] := -0.0304344;
   t5[2322] := -0.0298723;
   t5[2323] := -0.0293326;
   t5[2324] := -0.0288156;
   t5[2325] := -0.0283215;
   t5[2326] := -0.0278507;
   t5[2327] := -0.0274032;
   t5[2328] := -0.0269795;
   t5[2329] := -0.0265796;
   t5[2330] := -0.026204;
   t5[2331] := -0.0258527;
   t5[2332] := -0.0255261;
   t5[2333] := -0.0252244;
   t5[2334] := -0.0249478;
   t5[2335] := -0.0246962;
   t5[2336] := -0.0244691;
   t5[2337] := -0.0242663;
   t5[2338] := -0.0240873;
   t5[2339] := -0.0239318;
   t5[2340] := -0.0237993;
   t5[2341] := -0.0236896;
   t5[2342] := -0.0236022;
   t5[2343] := -0.0235369;
   t5[2344] := -0.0234931;
   t5[2345] := -0.0234706;
   t5[2346] := -0.0234689;
   t5[2347] := -0.0234878;
   t5[2348] := -0.0235268;
   t5[2349] := -0.0235855;
   t5[2350] := 0.0315658;
   t5[2351] := 0.0319544;
   t5[2352] := 0.0323323;
   t5[2353] := 0.0326995;
   t5[2354] := 0.033056;
   t5[2355] := 0.0334018;
   t5[2356] := 0.0337369;
   t5[2357] := 0.0340612;
   t5[2358] := 0.0343748;
   t5[2359] := 0.0346776;
   t5[2360] := 0.0349696;
   t5[2361] := 0.0352509;
   t5[2362] := 0.0355213;
   t5[2363] := 0.035781;
   t5[2364] := 0.0360298;
   t5[2365] := 0.0362678;
   t5[2366] := 0.0364949;
   t5[2367] := 0.0367111;
   t5[2368] := 0.0369165;
   t5[2369] := 0.037111;
   t5[2370] := 0.0372946;
   t5[2371] := 0.0374672;
   t5[2372] := 0.037629;
   t5[2373] := 0.0377798;
   t5[2374] := 0.0379196;
   t5[2375] := 0.0380485;
   t5[2376] := 0.0381664;
   t5[2377] := 0.0382733;
   t5[2378] := 0.0383692;
   t5[2379] := 0.0384541;
   t5[2380] := 0.0385279;
   t5[2381] := 0.0385907;
   t5[2382] := 0.0386425;
   t5[2383] := 0.0386832;
   t5[2384] := 0.0387128;
   t5[2385] := 0.0387315;
   t5[2386] := 0.0387396;
   t5[2387] := 0.0387371;
   t5[2388] := 0.0387245;
   t5[2389] := 0.0387019;
   t5[2390] := 0.0386695;
   t5[2391] := 0.0386276;
   t5[2392] := 0.0385764;
   t5[2393] := 0.0385161;
   t5[2394] := 0.038447;
   t5[2395] := 0.0383693;
   t5[2396] := 0.0382832;
   t5[2397] := 0.038189;
   t5[2398] := 0.038087;
   t5[2399] := 0.0379772;
   t5[2400] := 0.0589575;
   t5[2401] := 0.0584591;
   t5[2402] := 0.0579494;
   t5[2403] := 0.0574284;
   t5[2404] := 0.0568964;
   t5[2405] := 0.0563532;
   t5[2406] := 0.0557989;
   t5[2407] := 0.0552337;
   t5[2408] := 0.0546575;
   t5[2409] := 0.0540705;
   t5[2410] := 0.0534726;
   t5[2411] := 0.052864;
   t5[2412] := 0.0522447;
   t5[2413] := 0.0516147;
   t5[2414] := 0.0509741;
   t5[2415] := 0.050323;
   t5[2416] := 0.0496614;
   t5[2417] := 0.0489894;
   t5[2418] := 0.0483071;
   t5[2419] := 0.0476144;
   t5[2420] := 0.0469115;
   t5[2421] := 0.0461984;
   t5[2422] := 0.0454751;
   t5[2423] := 0.0447418;
   t5[2424] := 0.0439985;
   t5[2425] := 0.0432452;
   t5[2426] := 0.042482;
   t5[2427] := 0.041709;
   t5[2428] := 0.0409261;
   t5[2429] := 0.0401336;
   t5[2430] := 0.0393314;
   t5[2431] := 0.0385195;
   t5[2432] := 0.0376981;
   t5[2433] := 0.0368672;
   t5[2434] := 0.0360269;
   t5[2435] := 0.0351772;
   t5[2436] := 0.0343186;
   t5[2437] := 0.033451;
   t5[2438] := 0.0325749;
   t5[2439] := 0.0316903;
   t5[2440] := 0.0307976;
   t5[2441] := 0.0298968;
   t5[2442] := 0.0289883;
   t5[2443] := 0.0280723;
   t5[2444] := 0.0271489;
   t5[2445] := 0.0262184;
   t5[2446] := 0.025281;
   t5[2447] := 0.0243369;
   t5[2448] := 0.0233863;
   t5[2449] := 0.0224294;
   t5[2450] := -0.0370074;
   t5[2451] := -0.0362903;
   t5[2452] := -0.035563;
   t5[2453] := -0.0348254;
   t5[2454] := -0.0340776;
   t5[2455] := -0.0333193;
   t5[2456] := -0.0325505;
   t5[2457] := -0.0317711;
   t5[2458] := -0.0309811;
   t5[2459] := -0.0301802;
   t5[2460] := -0.0293685;
   t5[2461] := -0.0285458;
   t5[2462] := -0.0277121;
   t5[2463] := -0.0268673;
   t5[2464] := -0.0260112;
   t5[2465] := -0.0251437;
   t5[2466] := -0.0242649;
   t5[2467] := -0.0233745;
   t5[2468] := -0.0224726;
   t5[2469] := -0.021559;
   t5[2470] := -0.0206336;
   t5[2471] := -0.0196963;
   t5[2472] := -0.018747;
   t5[2473] := -0.0177857;
   t5[2474] := -0.0168123;
   t5[2475] := -0.0158266;
   t5[2476] := -0.0148286;
   t5[2477] := -0.0138181;
   t5[2478] := -0.0127952;
   t5[2479] := -0.0117597;
   t5[2480] := -0.0107114;
   t5[2481] := -0.0096504;
   t5[2482] := -0.0085765;
   t5[2483] := -0.0074897;
   t5[2484] := -0.0063898;
   t5[2485] := -0.005277;
   t5[2486] := -0.0041517;
   t5[2487] := -0.0030142;
   t5[2488] := -0.0018648;
   t5[2489] := -0.0007038;
   t5[2490] := 0.0004684;
   t5[2491] := 0.0016516;
   t5[2492] := 0.0028455;
   t5[2493] := 0.0040496;
   t5[2494] := 0.0052638;
   t5[2495] := 0.0064876;
   t5[2496] := 0.0077208;
   t5[2497] := 0.008963;
   t5[2498] := 0.010214;
   t5[2499] := 0.0114734;
   t5[2500] := -0.0503424;
   t5[2501] := -0.0518265;
   t5[2502] := -0.0533022;
   t5[2503] := -0.0547693;
   t5[2504] := -0.0562274;
   t5[2505] := -0.0576761;
   t5[2506] := -0.0591152;
   t5[2507] := -0.0605443;
   t5[2508] := -0.061963;
   t5[2509] := -0.063371;
   t5[2510] := -0.0647681;
   t5[2511] := -0.0661538;
   t5[2512] := -0.0675278;
   t5[2513] := -0.0688898;
   t5[2514] := -0.0702395;
   t5[2515] := -0.0715765;
   t5[2516] := -0.0729005;
   t5[2517] := -0.0742112;
   t5[2518] := -0.0755082;
   t5[2519] := -0.0767912;
   t5[2520] := -0.0780599;
   t5[2521] := -0.0793139;
   t5[2522] := -0.0805528;
   t5[2523] := -0.0817765;
   t5[2524] := -0.0829845;
   t5[2525] := -0.0841764;
   t5[2526] := -0.085352;
   t5[2527] := -0.086511;
   t5[2528] := -0.087653;
   t5[2529] := -0.0887776;
   t5[2530] := -0.0898846;
   t5[2531] := -0.0909735;
   t5[2532] := -0.0920441;
   t5[2533] := -0.0930961;
   t5[2534] := -0.0941291;
   t5[2535] := -0.095143;
   t5[2536] := -0.0961379;
   t5[2537] := -0.0971139;
   t5[2538] := -0.0980709;
   t5[2539] := -0.0990092;
   t5[2540] := -0.0999286;
   t5[2541] := -0.1008293;
   t5[2542] := -0.1017114;
   t5[2543] := -0.1025749;
   t5[2544] := -0.1034197;
   t5[2545] := -0.1042461;
   t5[2546] := -0.105054;
   t5[2547] := -0.1058436;
   t5[2548] := -0.1066147;
   t5[2549] := -0.1073677;
   t5[2550] := -0.1648159;
   t5[2551] := -0.1633702;
   t5[2552] := -0.1619071;
   t5[2553] := -0.1604269;
   t5[2554] := -0.15893;
   t5[2555] := -0.1574166;
   t5[2556] := -0.1558871;
   t5[2557] := -0.1543417;
   t5[2558] := -0.1527808;
   t5[2559] := -0.1512046;
   t5[2560] := -0.1496136;
   t5[2561] := -0.148008;
   t5[2562] := -0.1463881;
   t5[2563] := -0.1447542;
   t5[2564] := -0.1431066;
   t5[2565] := -0.1414457;
   t5[2566] := -0.1397718;
   t5[2567] := -0.1380851;
   t5[2568] := -0.1363861;
   t5[2569] := -0.1346749;
   t5[2570] := -0.1329519;
   t5[2571] := -0.1312175;
   t5[2572] := -0.1294719;
   t5[2573] := -0.1277154;
   t5[2574] := -0.1259484;
   t5[2575] := -0.1241712;
   t5[2576] := -0.122384;
   t5[2577] := -0.1205873;
   t5[2578] := -0.1187812;
   t5[2579] := -0.1169661;
   t5[2580] := -0.1151424;
   t5[2581] := -0.1133103;
   t5[2582] := -0.1114702;
   t5[2583] := -0.1096223;
   t5[2584] := -0.107767;
   t5[2585] := -0.1059046;
   t5[2586] := -0.1040352;
   t5[2587] := -0.1021592;
   t5[2588] := -0.1002768;
   t5[2589] := -0.0983883;
   t5[2590] := -0.096494;
   t5[2591] := -0.094594;
   t5[2592] := -0.0926887;
   t5[2593] := -0.0907782;
   t5[2594] := -0.088863;
   t5[2595] := -0.0869431;
   t5[2596] := -0.085019;
   t5[2597] := -0.0830908;
   t5[2598] := -0.0811587;
   t5[2599] := -0.0792232;
   t5[2600] := -0.0904827;
   t5[2601] := -0.0903118;
   t5[2602] := -0.090142;
   t5[2603] := -0.0899734;
   t5[2604] := -0.0898061;
   t5[2605] := -0.0896402;
   t5[2606] := -0.0894757;
   t5[2607] := -0.0893127;
   t5[2608] := -0.0891512;
   t5[2609] := -0.0889914;
   t5[2610] := -0.0888334;
   t5[2611] := -0.0886772;
   t5[2612] := -0.0885229;
   t5[2613] := -0.0883705;
   t5[2614] := -0.0882202;
   t5[2615] := -0.0880719;
   t5[2616] := -0.0879259;
   t5[2617] := -0.0877822;
   t5[2618] := -0.0876408;
   t5[2619] := -0.0875018;
   t5[2620] := -0.0873653;
   t5[2621] := -0.0872314;
   t5[2622] := -0.0871001;
   t5[2623] := -0.0869716;
   t5[2624] := -0.0868459;
   t5[2625] := -0.086723;
   t5[2626] := -0.0866031;
   t5[2627] := -0.0864863;
   t5[2628] := -0.0863725;
   t5[2629] := -0.0862619;
   t5[2630] := -0.0861546;
   t5[2631] := -0.0860506;
   t5[2632] := -0.0859501;
   t5[2633] := -0.085853;
   t5[2634] := -0.0857595;
   t5[2635] := -0.0856695;
   t5[2636] := -0.0855828;
   t5[2637] := -0.0854994;
   t5[2638] := -0.0854192;
   t5[2639] := -0.085342;
   t5[2640] := -0.0852676;
   t5[2641] := -0.0851961;
   t5[2642] := -0.0851272;
   t5[2643] := -0.0850608;
   t5[2644] := -0.0849969;
   t5[2645] := -0.0849353;
   t5[2646] := -0.0848758;
   t5[2647] := -0.0848184;
   t5[2648] := -0.084763;
   t5[2649] := -0.0847093;
   t5[2650] := -0.0673839;
   t5[2651] := -0.066065;
   t5[2652] := -0.0647407;
   t5[2653] := -0.0634112;
   t5[2654] := -0.0620767;
   t5[2655] := -0.0607376;
   t5[2656] := -0.059394;
   t5[2657] := -0.0580462;
   t5[2658] := -0.0566946;
   t5[2659] := -0.0553392;
   t5[2660] := -0.0539806;
   t5[2661] := -0.0526187;
   t5[2662] := -0.0512541;
   t5[2663] := -0.0498868;
   t5[2664] := -0.0485171;
   t5[2665] := -0.0471454;
   t5[2666] := -0.0457718;
   t5[2667] := -0.0443967;
   t5[2668] := -0.0430202;
   t5[2669] := -0.0416427;
   t5[2670] := -0.0402645;
   t5[2671] := -0.0388857;
   t5[2672] := -0.0375066;
   t5[2673] := -0.0361275;
   t5[2674] := -0.0347487;
   t5[2675] := -0.0333704;
   t5[2676] := -0.0319928;
   t5[2677] := -0.0306163;
   t5[2678] := -0.0292411;
   t5[2679] := -0.0278674;
   t5[2680] := -0.0264955;
   t5[2681] := -0.0251257;
   t5[2682] := -0.0237583;
   t5[2683] := -0.0223934;
   t5[2684] := -0.0210313;
   t5[2685] := -0.0196723;
   t5[2686] := -0.0183165;
   t5[2687] := -0.0169639;
   t5[2688] := -0.0156148;
   t5[2689] := -0.0142693;
   t5[2690] := -0.0129275;
   t5[2691] := -0.0115895;
   t5[2692] := -0.0102555;
   t5[2693] := -0.0089257;
   t5[2694] := -0.0076001;
   t5[2695] := -0.006279;
   t5[2696] := -0.0049623;
   t5[2697] := -0.0036504;
   t5[2698] := -0.0023433;
   t5[2699] := -0.0010412;
   t5[2700] := 0.075334;
   t5[2701] := 0.0752603;
   t5[2702] := 0.0751656;
   t5[2703] := 0.0750495;
   t5[2704] := 0.0749118;
   t5[2705] := 0.0747521;
   t5[2706] := 0.0745704;
   t5[2707] := 0.0743661;
   t5[2708] := 0.0741392;
   t5[2709] := 0.0738893;
   t5[2710] := 0.0736161;
   t5[2711] := 0.0733193;
   t5[2712] := 0.0729987;
   t5[2713] := 0.072654;
   t5[2714] := 0.072285;
   t5[2715] := 0.0718913;
   t5[2716] := 0.0714727;
   t5[2717] := 0.0710288;
   t5[2718] := 0.0705595;
   t5[2719] := 0.0700644;
   t5[2720] := 0.0695434;
   t5[2721] := 0.068996;
   t5[2722] := 0.068422;
   t5[2723] := 0.0678212;
   t5[2724] := 0.0671932;
   t5[2725] := 0.0665378;
   t5[2726] := 0.0658548;
   t5[2727] := 0.0651437;
   t5[2728] := 0.0644045;
   t5[2729] := 0.0636367;
   t5[2730] := 0.0628402;
   t5[2731] := 0.0620146;
   t5[2732] := 0.0611596;
   t5[2733] := 0.0602751;
   t5[2734] := 0.0593606;
   t5[2735] := 0.0584166;
   t5[2736] := 0.0574435;
   t5[2737] := 0.0564417;
   t5[2738] := 0.0554119;
   t5[2739] := 0.0543544;
   t5[2740] := 0.0532698;
   t5[2741] := 0.0521586;
   t5[2742] := 0.0510212;
   t5[2743] := 0.0498582;
   t5[2744] := 0.0486701;
   t5[2745] := 0.0474574;
   t5[2746] := 0.0462205;
   t5[2747] := 0.04496;
   t5[2748] := 0.0436763;
   t5[2749] := 0.04237;
   t5[2750] := -0.1063465;
   t5[2751] := -0.1058427;
   t5[2752] := -0.105332;
   t5[2753] := -0.1048147;
   t5[2754] := -0.1042907;
   t5[2755] := -0.1037601;
   t5[2756] := -0.1032231;
   t5[2757] := -0.1026798;
   t5[2758] := -0.1021301;
   t5[2759] := -0.1015743;
   t5[2760] := -0.1010124;
   t5[2761] := -0.1004444;
   t5[2762] := -0.0998706;
   t5[2763] := -0.0992909;
   t5[2764] := -0.0987055;
   t5[2765] := -0.0981145;
   t5[2766] := -0.0975178;
   t5[2767] := -0.0969158;
   t5[2768] := -0.0963083;
   t5[2769] := -0.0956956;
   t5[2770] := -0.0950776;
   t5[2771] := -0.0944546;
   t5[2772] := -0.0938265;
   t5[2773] := -0.0931935;
   t5[2774] := -0.0925557;
   t5[2775] := -0.0919131;
   t5[2776] := -0.0912658;
   t5[2777] := -0.090614;
   t5[2778] := -0.0899577;
   t5[2779] := -0.089297;
   t5[2780] := -0.088632;
   t5[2781] := -0.0879628;
   t5[2782] := -0.0872895;
   t5[2783] := -0.0866122;
   t5[2784] := -0.0859309;
   t5[2785] := -0.0852457;
   t5[2786] := -0.0845565;
   t5[2787] := -0.0838635;
   t5[2788] := -0.0831666;
   t5[2789] := -0.0824658;
   t5[2790] := -0.0817611;
   t5[2791] := -0.0810525;
   t5[2792] := -0.0803401;
   t5[2793] := -0.0796237;
   t5[2794] := -0.0789035;
   t5[2795] := -0.0781795;
   t5[2796] := -0.0774516;
   t5[2797] := -0.0767199;
   t5[2798] := -0.0759843;
   t5[2799] := -0.0752448;
   t5[2800] := 0.0025241;
   t5[2801] := 0.0019133;
   t5[2802] := 0.0012993;
   t5[2803] := 0.0006824;
   t5[2804] := 6.28E-05;
   t5[2805] := -0.0005596;
   t5[2806] := -0.0011845;
   t5[2807] := -0.0018117;
   t5[2808] := -0.0024413;
   t5[2809] := -0.003073;
   t5[2810] := -0.0037067;
   t5[2811] := -0.0043423;
   t5[2812] := -0.0049797;
   t5[2813] := -0.0056187;
   t5[2814] := -0.0062591;
   t5[2815] := -0.006901;
   t5[2816] := -0.0075441;
   t5[2817] := -0.0081882;
   t5[2818] := -0.0088334;
   t5[2819] := -0.0094794;
   t5[2820] := -0.0101261;
   t5[2821] := -0.0107734;
   t5[2822] := -0.0114211;
   t5[2823] := -0.0120691;
   t5[2824] := -0.0127174;
   t5[2825] := -0.0133657;
   t5[2826] := -0.0140139;
   t5[2827] := -0.014662;
   t5[2828] := -0.0153097;
   t5[2829] := -0.0159569;
   t5[2830] := -0.0166036;
   t5[2831] := -0.0172495;
   t5[2832] := -0.0178946;
   t5[2833] := -0.0185387;
   t5[2834] := -0.0191817;
   t5[2835] := -0.0198235;
   t5[2836] := -0.0204642;
   t5[2837] := -0.0211037;
   t5[2838] := -0.0217419;
   t5[2839] := -0.0223789;
   t5[2840] := -0.0230147;
   t5[2841] := -0.0236492;
   t5[2842] := -0.0242824;
   t5[2843] := -0.0249143;
   t5[2844] := -0.0255448;
   t5[2845] := -0.0261741;
   t5[2846] := -0.0268019;
   t5[2847] := -0.0274284;
   t5[2848] := -0.0280535;
   t5[2849] := -0.0286772;
   t5[2850] := -0.0587365;
   t5[2851] := -0.0607911;
   t5[2852] := -0.0628394;
   t5[2853] := -0.0648808;
   t5[2854] := -0.0669146;
   t5[2855] := -0.0689402;
   t5[2856] := -0.0709572;
   t5[2857] := -0.0729648;
   t5[2858] := -0.0749626;
   t5[2859] := -0.0769499;
   t5[2860] := -0.0789262;
   t5[2861] := -0.0808909;
   t5[2862] := -0.0828433;
   t5[2863] := -0.084783;
   t5[2864] := -0.0867094;
   t5[2865] := -0.0886217;
   t5[2866] := -0.0905196;
   t5[2867] := -0.0924023;
   t5[2868] := -0.0942693;
   t5[2869] := -0.09612;
   t5[2870] := -0.0979539;
   t5[2871] := -0.0997704;
   t5[2872] := -0.1015688;
   t5[2873] := -0.1033487;
   t5[2874] := -0.1051093;
   t5[2875] := -0.1068502;
   t5[2876] := -0.1085707;
   t5[2877] := -0.1102703;
   t5[2878] := -0.1119484;
   t5[2879] := -0.1136044;
   t5[2880] := -0.1152377;
   t5[2881] := -0.1168477;
   t5[2882] := -0.1184339;
   t5[2883] := -0.1199957;
   t5[2884] := -0.1215325;
   t5[2885] := -0.1230443;
   t5[2886] := -0.1245312;
   t5[2887] := -0.1259933;
   t5[2888] := -0.1274307;
   t5[2889] := -0.1288437;
   t5[2890] := -0.1302324;
   t5[2891] := -0.1315969;
   t5[2892] := -0.1329374;
   t5[2893] := -0.134254;
   t5[2894] := -0.1355468;
   t5[2895] := -0.1368162;
   t5[2896] := -0.138062;
   t5[2897] := -0.1392847;
   t5[2898] := -0.1404841;
   t5[2899] := -0.1416606;
   t5[2900] := -0.0241061;
   t5[2901] := -0.0237218;
   t5[2902] := -0.0233311;
   t5[2903] := -0.0229339;
   t5[2904] := -0.0225301;
   t5[2905] := -0.0221195;
   t5[2906] := -0.021702;
   t5[2907] := -0.0212774;
   t5[2908] := -0.0208456;
   t5[2909] := -0.0204065;
   t5[2910] := -0.0199598;
   t5[2911] := -0.0195055;
   t5[2912] := -0.0190435;
   t5[2913] := -0.0185735;
   t5[2914] := -0.0180954;
   t5[2915] := -0.0176091;
   t5[2916] := -0.0171145;
   t5[2917] := -0.0166113;
   t5[2918] := -0.0160995;
   t5[2919] := -0.015579;
   t5[2920] := -0.0150495;
   t5[2921] := -0.0145109;
   t5[2922] := -0.0139632;
   t5[2923] := -0.0134061;
   t5[2924] := -0.0128394;
   t5[2925] := -0.0122632;
   t5[2926] := -0.0116771;
   t5[2927] := -0.0110811;
   t5[2928] := -0.0104751;
   t5[2929] := -0.0098588;
   t5[2930] := -0.0092322;
   t5[2931] := -0.0085951;
   t5[2932] := -0.0079474;
   t5[2933] := -0.0072889;
   t5[2934] := -0.0066194;
   t5[2935] := -0.0059392;
   t5[2936] := -0.0052484;
   t5[2937] := -0.0045472;
   t5[2938] := -0.003836;
   t5[2939] := -0.0031149;
   t5[2940] := -0.0023841;
   t5[2941] := -0.001644;
   t5[2942] := -0.0008946;
   t5[2943] := -0.0001363;
   t5[2944] := 0.0006307;
   t5[2945] := 0.0014062;
   t5[2946] := 0.0021899;
   t5[2947] := 0.0029816;
   t5[2948] := 0.0037812;
   t5[2949] := 0.0045883;
   t5[2950] := -0.016338;
   t5[2951] := -0.0155328;
   t5[2952] := -0.0147281;
   t5[2953] := -0.013924;
   t5[2954] := -0.0131203;
   t5[2955] := -0.012317;
   t5[2956] := -0.0115141;
   t5[2957] := -0.0107115;
   t5[2958] := -0.009909;
   t5[2959] := -0.0091068;
   t5[2960] := -0.0083047;
   t5[2961] := -0.0075027;
   t5[2962] := -0.0067006;
   t5[2963] := -0.0058985;
   t5[2964] := -0.0050963;
   t5[2965] := -0.0042939;
   t5[2966] := -0.0034913;
   t5[2967] := -0.0026884;
   t5[2968] := -0.0018852;
   t5[2969] := -0.0010816;
   t5[2970] := -0.0002775;
   t5[2971] := 0.0005271;
   t5[2972] := 0.0013323;
   t5[2973] := 0.0021381;
   t5[2974] := 0.0029446;
   t5[2975] := 0.0037519;
   t5[2976] := 0.0045599;
   t5[2977] := 0.0053689;
   t5[2978] := 0.0061787;
   t5[2979] := 0.0069895;
   t5[2980] := 0.0078014;
   t5[2981] := 0.0086143;
   t5[2982] := 0.0094284;
   t5[2983] := 0.0102437;
   t5[2984] := 0.0110602;
   t5[2985] := 0.011878;
   t5[2986] := 0.0126969;
   t5[2987] := 0.0135169;
   t5[2988] := 0.0143378;
   t5[2989] := 0.0151596;
   t5[2990] := 0.0159821;
   t5[2991] := 0.0168054;
   t5[2992] := 0.0176293;
   t5[2993] := 0.0184537;
   t5[2994] := 0.0192785;
   t5[2995] := 0.0201037;
   t5[2996] := 0.0209292;
   t5[2997] := 0.0217548;
   t5[2998] := 0.0225805;
   t5[2999] := 0.0234063;
   t5[3000] := -0.0519279;
   t5[3001] := -0.053238;
   t5[3002] := -0.054539;
   t5[3003] := -0.0558307;
   t5[3004] := -0.0571129;
   t5[3005] := -0.0583854;
   t5[3006] := -0.059648;
   t5[3007] := -0.0609004;
   t5[3008] := -0.0621425;
   t5[3009] := -0.0633741;
   t5[3010] := -0.0645949;
   t5[3011] := -0.0658048;
   t5[3012] := -0.0670035;
   t5[3013] := -0.0681909;
   t5[3014] := -0.0693667;
   t5[3015] := -0.0705308;
   t5[3016] := -0.0716829;
   t5[3017] := -0.0728229;
   t5[3018] := -0.0739505;
   t5[3019] := -0.0750655;
   t5[3020] := -0.0761677;
   t5[3021] := -0.0772569;
   t5[3022] := -0.078333;
   t5[3023] := -0.0793957;
   t5[3024] := -0.0804448;
   t5[3025] := -0.08148;
   t5[3026] := -0.0825013;
   t5[3027] := -0.0835084;
   t5[3028] := -0.0845011;
   t5[3029] := -0.0854791;
   t5[3030] := -0.0864423;
   t5[3031] := -0.0873905;
   t5[3032] := -0.0883235;
   t5[3033] := -0.0892411;
   t5[3034] := -0.090143;
   t5[3035] := -0.0910294;
   t5[3036] := -0.0919002;
   t5[3037] := -0.0927557;
   t5[3038] := -0.093596;
   t5[3039] := -0.0944211;
   t5[3040] := -0.0952312;
   t5[3041] := -0.0960264;
   t5[3042] := -0.0968068;
   t5[3043] := -0.0975726;
   t5[3044] := -0.0983239;
   t5[3045] := -0.0990608;
   t5[3046] := -0.0997833;
   t5[3047] := -0.1004917;
   t5[3048] := -0.101186;
   t5[3049] := -0.1018665;
   t5[3050] := 0.142846;
   t5[3051] := 0.1421979;
   t5[3052] := 0.1415383;
   t5[3053] := 0.1408671;
   t5[3054] := 0.1401842;
   t5[3055] := 0.1394896;
   t5[3056] := 0.1387834;
   t5[3057] := 0.1380653;
   t5[3058] := 0.1373355;
   t5[3059] := 0.1365938;
   t5[3060] := 0.1358403;
   t5[3061] := 0.1350748;
   t5[3062] := 0.1342974;
   t5[3063] := 0.133508;
   t5[3064] := 0.1327065;
   t5[3065] := 0.131893;
   t5[3066] := 0.1310673;
   t5[3067] := 0.1302295;
   t5[3068] := 0.1293795;
   t5[3069] := 0.1285172;
   t5[3070] := 0.1276427;
   t5[3071] := 0.1267559;
   t5[3072] := 0.1258567;
   t5[3073] := 0.124945;
   t5[3074] := 0.124021;
   t5[3075] := 0.1230845;
   t5[3076] := 0.1221354;
   t5[3077] := 0.1211738;
   t5[3078] := 0.1201996;
   t5[3079] := 0.1192127;
   t5[3080] := 0.1182132;
   t5[3081] := 0.1172009;
   t5[3082] := 0.1161759;
   t5[3083] := 0.1151381;
   t5[3084] := 0.1140875;
   t5[3085] := 0.1130242;
   t5[3086] := 0.1119484;
   t5[3087] := 0.1108604;
   t5[3088] := 0.1097604;
   t5[3089] := 0.1086486;
   t5[3090] := 0.1075254;
   t5[3091] := 0.1063909;
   t5[3092] := 0.1052453;
   t5[3093] := 0.1040889;
   t5[3094] := 0.1029219;
   t5[3095] := 0.1017446;
   t5[3096] := 0.1005571;
   t5[3097] := 0.0993598;
   t5[3098] := 0.0981528;
   t5[3099] := 0.0969364;
   t5[3100] := -0.0299947;
   t5[3101] := -0.0298427;
   t5[3102] := -0.0296883;
   t5[3103] := -0.0295314;
   t5[3104] := -0.029372;
   t5[3105] := -0.0292101;
   t5[3106] := -0.0290456;
   t5[3107] := -0.0288785;
   t5[3108] := -0.0287087;
   t5[3109] := -0.0285362;
   t5[3110] := -0.028361;
   t5[3111] := -0.028183;
   t5[3112] := -0.0280021;
   t5[3113] := -0.0278184;
   t5[3114] := -0.0276319;
   t5[3115] := -0.0274423;
   t5[3116] := -0.0272498;
   t5[3117] := -0.0270543;
   t5[3118] := -0.0268557;
   t5[3119] := -0.026654;
   t5[3120] := -0.0264491;
   t5[3121] := -0.0262411;
   t5[3122] := -0.0260299;
   t5[3123] := -0.0258154;
   t5[3124] := -0.0255976;
   t5[3125] := -0.0253764;
   t5[3126] := -0.0251519;
   t5[3127] := -0.024924;
   t5[3128] := -0.0246926;
   t5[3129] := -0.0244577;
   t5[3130] := -0.0242193;
   t5[3131] := -0.0239773;
   t5[3132] := -0.0237317;
   t5[3133] := -0.0234824;
   t5[3134] := -0.0232294;
   t5[3135] := -0.0229728;
   t5[3136] := -0.0227127;
   t5[3137] := -0.0224492;
   t5[3138] := -0.0221823;
   t5[3139] := -0.0219122;
   t5[3140] := -0.021639;
   t5[3141] := -0.0213628;
   t5[3142] := -0.0210837;
   t5[3143] := -0.0208018;
   t5[3144] := -0.0205172;
   t5[3145] := -0.0202301;
   t5[3146] := -0.0199404;
   t5[3147] := -0.0196484;
   t5[3148] := -0.019354;
   t5[3149] := -0.0190576;
   t5[3150] := -0.0100999;
   t5[3151] := -0.008071;
   t5[3152] := -0.0060584;
   t5[3153] := -0.0040626;
   t5[3154] := -0.0020842;
   t5[3155] := -0.0001238;
   t5[3156] := 0.001818;
   t5[3157] := 0.0037406;
   t5[3158] := 0.0056435;
   t5[3159] := 0.007526;
   t5[3160] := 0.0093876;
   t5[3161] := 0.0112276;
   t5[3162] := 0.0130455;
   t5[3163] := 0.0148407;
   t5[3164] := 0.0166126;
   t5[3165] := 0.0183606;
   t5[3166] := 0.0200841;
   t5[3167] := 0.0217825;
   t5[3168] := 0.0234553;
   t5[3169] := 0.0251017;
   t5[3170] := 0.0267214;
   t5[3171] := 0.0283136;
   t5[3172] := 0.0298777;
   t5[3173] := 0.0314133;
   t5[3174] := 0.0329196;
   t5[3175] := 0.0343962;
   t5[3176] := 0.0358423;
   t5[3177] := 0.0372574;
   t5[3178] := 0.038641;
   t5[3179] := 0.0399924;
   t5[3180] := 0.0413111;
   t5[3181] := 0.0425964;
   t5[3182] := 0.0438478;
   t5[3183] := 0.0450646;
   t5[3184] := 0.0462464;
   t5[3185] := 0.0473932;
   t5[3186] := 0.0485056;
   t5[3187] := 0.0495838;
   t5[3188] := 0.0506283;
   t5[3189] := 0.0516397;
   t5[3190] := 0.0526183;
   t5[3191] := 0.0535646;
   t5[3192] := 0.054479;
   t5[3193] := 0.055362;
   t5[3194] := 0.0562139;
   t5[3195] := 0.0570354;
   t5[3196] := 0.0578267;
   t5[3197] := 0.0585883;
   t5[3198] := 0.0593207;
   t5[3199] := 0.0600244;
   w6[0] := 0.0254122;
   w6[1] := -0.4251655;
   w6[2] := -0.4513899;
   w6[3] := 0.0262705;
   w6[4] := 0.3702881;
   w6[5] := -0.1208161;
   w6[6] := -0.2231239;
   w6[7] := 0.2512441;
   w6[8] := -0.3278799;
   w6[9] := 0.2889541;
   w6[10] := -0.0654242;
   w6[11] := 0.1067281;
   w6[12] := 0.2623815;
   w6[13] := -0.1798091;
   w6[14] := -0.3070911;
   w6[15] := -0.4204447;
   w6[16] := 0.5762351;
   w6[17] := -1.090657;
   w6[18] := -0.2690518;
   w6[19] := -0.6730261;
   w6[20] := -0.0514923;
   w6[21] := -0.4457789;
   w6[22] := 0.5072183;
   w6[23] := -0.0549661;
   w6[24] := 0.3812394;
   w6[25] := -0.606307;
   w6[26] := 0.1917919;
   w6[27] := 0.1525442;
   w6[28] := -0.4219312;
   w6[29] := 0.338313;
   w6[30] := 0.1919874;
   w6[31] := -0.3457294;
   w6[32] := 0.1728978;
   w6[33] := 0.5825878;
   w6[34] := 0.7331663;
   w6[35] := 0.4268312;
   w6[36] := -0.0077422;
   w6[37] := 0.4766487;
   w6[38] := 0.102607;
   w6[39] := -0.5723706;
   w6[40] := 0.0728498;
   w6[41] := 0.4253429;
   w6[42] := -0.3637053;
   w6[43] := -0.6206156;
   w6[44] := 0.2656944;
   w6[45] := -0.3130539;
   w6[46] := 0.2033212;
   w6[47] := 0.1327122;
   w6[48] := -0.709101;
   w6[49] := 0.7231103;
   w6[50] := -0.2214241;
   w6[51] := 0.4491622;
   w6[52] := -0.3655713;
   w6[53] := 0.4263724;
   w6[54] := 0.0266531;
   w6[55] := 0.4637966;
   w6[56] := -0.3418979;
   w6[57] := -0.2391363;
   w6[58] := 0.4152579;
   w6[59] := 0.2146362;
   w6[60] := -0.3901598;
   w6[61] := -0.1938754;
   w6[62] := -0.561949;
   w6[63] := 0.4047181;
END_DATA_BLOCK

FUNCTION_BLOCK "NeuroPLC_Inference"   // FB1, SCL
{ S7_Optimized_Access := 'FALSE' }
VERSION : 0.1
// NeuroPLC 鈥?Auto-generated IEC 61131-3 SCL (DB+FB Mode)
//  Graph: kan | Target: S71500DBBackend
//  Work memory: 1500KB | LUT points: 50
//  Nodes: 11 | Ops: {'matmul': 3, 'standard_act': 2, 'bspline_lut': 2, 'add': 2, 'softmax': 1, 'argmax': 1}
//  Parameters in DB "NeuroPLC_KAN_Weights", inference in FB.
   VAR_INPUT
      features : Array[0..27] of Real;   // 28-D feature vector
   END_VAR
   VAR_OUTPUT
      fault_class : Int;   // 0=Normal, 1=InnerRace, 2=Ball, 3=OuterRace
      confidence : Real;   // max softmax probability 鈹€鈹€ Inference temporaries 鈹€鈹€
   END_VAR
   VAR
      v1 : Array[0..27] of Real;   // silu output
      v3 : Array[0..447] of Real;   // BsplineLUT output (1D: o*28+i)
      v2 : Array[0..15] of Real;   // matmul output
      v4 : Array[0..15] of Real;   // add merge
      v5 : Array[0..15] of Real;   // silu output
      v7 : Array[0..63] of Real;   // BsplineLUT output (1D: o*16+i)
      v6 : Array[0..3] of Real;   // matmul output
      v8 : Array[0..3] of Real;   // add merge
      v9 : Array[0..3] of Real;   // softmax output 鈹€鈹€ Temporary variables 鈹€鈹€
      i : Int;
      o : Int;
      j : Int;
      lo : Int;
      hi : Int;
      idx : Int;
      base : Int;
      sum : Real;
      max_val : Real;
      t_val : Real;
   END_VAR
BEGIN
      // 鈺愨晲鈺?Inference forward pass 鈺愨晲鈺?
       // Parameters loaded from DB "NeuroPLC_KAN_Weights" (start values = data, not code)

          // Input: features[0..27]

          // StandardAct: silu
          FOR #i := 0 TO 27 DO
              // SiLU = x / (1 + exp(-x))
              #v1[#i] := #features[#i] / (1.0 + EXP(-#features[#i]));
          END_FOR;

